LIN {X 0,Y 600.073,Z 913.37,A -85,B 0,C 180,E1 9120.834,E2 9120.834} C_VEL
LIN {X 0,Y 603.97,Z 872.465,A -85,B 0,C 180,E1 9122.572,E2 9122.572} C_VEL
LIN {X 0,Y 605.713,Z 840.651,A -85,B 0,C 180,E1 9123.575,E2 9123.575} C_VEL
LIN {X 0,Y 586.548,Z 799.806,A -85,B 0,C 180,E1 9125.931,E2 9125.931} C_VEL
LIN {X 0,Y 577.288,Z 782.326,A -85,B 0,C 180,E1 9126.944,E2 9126.944} C_VEL
LIN {X 0,Y 577.109,Z 780.81,A -85,B 0,C 180,E1 9127.031,E2 9127.031} C_VEL
LIN {X 0,Y 577.142,Z 780.81,A -85,B 0,C 180,E1 9132.903,E2 9132.903} C_VEL
LIN {X 0,Y 577.108,Z 780.81,A -85,B 0,C 180,E1 9139.116,E2 9139.116} C_VEL
LIN {X 0,Y 577.097,Z 780.81,A -85,B 0,C 180,E1 9144.83,E2 9144.83} C_VEL
LIN {X 0,Y 577.255,Z 780.81,A -85,B 0,C 180,E1 9150.177,E2 9150.177} C_VEL
LIN {X 0,Y 577.406,Z 780.81,A -85,B 0,C 180,E1 9155.248,E2 9155.248} C_VEL
LIN {X 0,Y 577.552,Z 780.81,A -85,B 0,C 180,E1 9160.376,E2 9160.376} C_VEL
LIN {X 0,Y 577.609,Z 780.81,A -85,B 0,C 180,E1 9165.463,E2 9165.463} C_VEL
LIN {X 0,Y 577.862,Z 780.81,A -85,B 0,C 180,E1 9170.972,E2 9170.972} C_VEL
LIN {X 0,Y 578.107,Z 780.81,A -85,B 0,C 180,E1 9177.002,E2 9177.002} C_VEL
LIN {X 0,Y 578.174,Z 780.81,A -85,B 0,C 180,E1 9181.495,E2 9181.495} C_VEL
LIN {X 0,Y 577.898,Z 780.81,A -85,B 0,C 180,E1 9187.509,E2 9187.509} C_VEL
LIN {X 0,Y 577.695,Z 780.81,A -85,B 0,C 180,E1 9193.611,E2 9193.611} C_VEL
LIN {X 0,Y 577.587,Z 780.81,A -85,B 0,C 180,E1 9199.634,E2 9199.634} C_VEL
LIN {X 0,Y 577.399,Z 780.81,A -85,B 0,C 180,E1 9204.748,E2 9204.748} C_VEL
LIN {X 0,Y 577.283,Z 780.81,A -85,B 0,C 180,E1 9210.251,E2 9210.251} C_VEL
LIN {X 0,Y 577.16,Z 780.81,A -85,B 0,C 180,E1 9215.743,E2 9215.743} C_VEL
LIN {X 0,Y 577.065,Z 780.81,A -85,B 0,C 180,E1 9220.882,E2 9220.882} C_VEL
LIN {X 0,Y 577.059,Z 780.81,A -85,B 0,C 180,E1 9227.143,E2 9227.143} C_VEL
LIN {X 0,Y 577.082,Z 780.895,A -85,B 0,C 180,E1 9229.475,E2 9229.475} C_VEL
LIN {X 0,Y 581.683,Z 790.937,A -85,B 0,C 180,E1 9230,E2 9230} C_VEL
LIN {X 0,Y 607.436,Z 841.355,A -85,B 0,C 180,E1 9232.688,E2 9232.688} C_VEL
LIN {X 0,Y 605.125,Z 884.485,A -85,B 0,C 180,E1 9233.623,E2 9233.623} C_VEL
LIN {X 0,Y 604.334,Z 895.912,A -85,B 0,C 180,E1 9233.955,E2 9233.955} C_VEL
LIN {X 0,Y 599.805,Z 912.465,A -85,B 0,C 180,E1 9234.299,E2 9234.299} C_VEL
LIN {X 0,Y 594.958,Z 928.635,A -85,B 0,C 180,E1 9234.736,E2 9234.736} C_VEL
LIN {X 0,Y 590.175,Z 971.895,A -85,B 0,C 180,E1 9236.914,E2 9236.914} C_VEL
LIN {X 0,Y 585.078,Z 1013.237,A -85,B 0,C 180,E1 9239.768,E2 9239.768} C_VEL
LIN {X 0,Y 580.557,Z 1047.846,A -85,B 0,C 180,E1 9242.902,E2 9242.902} C_VEL
LIN {X 0,Y 576.578,Z 1078.993,A -85,B 0,C 180,E1 9246.504,E2 9246.504} C_VEL
LIN {X 0,Y 573.684,Z 1106.248,A -85,B 0,C 180,E1 9250.576,E2 9250.576} C_VEL
LIN {X 0,Y 571.664,Z 1128.837,A -85,B 0,C 180,E1 9255.064,E2 9255.064} C_VEL
LIN {X 0,Y 570.638,Z 1145.24,A -85,B 0,C 180,E1 9259.702,E2 9259.702} C_VEL
LIN {X 0,Y 570.381,Z 1154.482,A -85,B 0,C 180,E1 9263.916,E2 9263.916} C_VEL
LIN {X 0,Y 570.304,Z 1159.165,A -85,B 0,C 180,E1 9268.481,E2 9268.481} C_VEL
LIN {X 0,Y 570.212,Z 1158.218,A -85,B 0,C 180,E1 9273.037,E2 9273.037} C_VEL
LIN {X 0,Y 570.422,Z 1152.885,A -85,B 0,C 180,E1 9277.02,E2 9277.02} C_VEL
LIN {X 0,Y 570.84,Z 1142.468,A -85,B 0,C 180,E1 9281.212,E2 9281.212} C_VEL
LIN {X 0,Y 571.852,Z 1127.098,A -85,B 0,C 180,E1 9285.321,E2 9285.321} C_VEL
LIN {X 0,Y 573.818,Z 1105.125,A -85,B 0,C 180,E1 9289.618,E2 9289.618} C_VEL
LIN {X 0,Y 576.919,Z 1076.481,A -85,B 0,C 180,E1 9293.824,E2 9293.824} C_VEL
LIN {X 0,Y 581.055,Z 1043.921,A -85,B 0,C 180,E1 9297.49,E2 9297.49} C_VEL
LIN {X 0,Y 585.633,Z 1008.232,A -85,B 0,C 180,E1 9300.619,E2 9300.619} C_VEL
LIN {X 0,Y 590.548,Z 969.141,A -85,B 0,C 180,E1 9303.259,E2 9303.259} C_VEL
LIN {X 0,Y 595.375,Z 925.534,A -85,B 0,C 180,E1 9305.435,E2 9305.435} C_VEL
LIN {X 0,Y 599.416,Z 879.277,A -85,B 0,C 180,E1 9307.007,E2 9307.007} C_VEL
LIN {X 0,Y 601.018,Z 843.241,A -85,B 0,C 180,E1 9307.816,E2 9307.816} C_VEL
LIN {X 0,Y 580.212,Z 801.744,A -85,B 0,C 180,E1 9310.177,E2 9310.177} C_VEL
LIN {X 0,Y 569.244,Z 781.517,A -85,B 0,C 180,E1 9311.481,E2 9311.481} C_VEL
LIN {X 0,Y 569.183,Z 780.81,A -85,B 0,C 180,E1 9316.362,E2 9316.362} C_VEL
LIN {X 0,Y 569.222,Z 780.81,A -85,B 0,C 180,E1 9322.379,E2 9322.379} C_VEL
LIN {X 0,Y 569.268,Z 780.81,A -85,B 0,C 180,E1 9328.148,E2 9328.148} C_VEL
LIN {X 0,Y 569.463,Z 780.81,A -85,B 0,C 180,E1 9333.193,E2 9333.193} C_VEL
LIN {X 0,Y 569.555,Z 780.81,A -85,B 0,C 180,E1 9338.215,E2 9338.215} C_VEL
LIN {X 0,Y 569.678,Z 780.81,A -85,B 0,C 180,E1 9343.041,E2 9343.041} C_VEL
LIN {X 0,Y 569.786,Z 780.81,A -85,B 0,C 180,E1 9348.886,E2 9348.886} C_VEL
LIN {X 0,Y 569.989,Z 780.81,A -85,B 0,C 180,E1 9353.916,E2 9353.916} C_VEL
LIN {X 0,Y 570.111,Z 780.81,A -85,B 0,C 180,E1 9358.484,E2 9358.484} C_VEL
LIN {X 0,Y 570.061,Z 780.81,A -85,B 0,C 180,E1 9363.041,E2 9363.041} C_VEL
LIN {X 0,Y 569.988,Z 780.81,A -85,B 0,C 180,E1 9367.618,E2 9367.618} C_VEL
LIN {X 0,Y 569.809,Z 780.81,A -85,B 0,C 180,E1 9372.249,E2 9372.249} C_VEL
LIN {X 0,Y 569.676,Z 780.81,A -85,B 0,C 180,E1 9377.271,E2 9377.271} C_VEL
LIN {X 0,Y 569.524,Z 780.81,A -85,B 0,C 180,E1 9381.804,E2 9381.804} C_VEL
LIN {X 0,Y 569.41,Z 780.81,A -85,B 0,C 180,E1 9386.815,E2 9386.815} C_VEL
LIN {X 0,Y 569.307,Z 780.81,A -85,B 0,C 180,E1 9392.06,E2 9392.06} C_VEL
LIN {X 0,Y 569.177,Z 780.81,A -85,B 0,C 180,E1 9397.63,E2 9397.63} C_VEL
LIN {X 0,Y 569.148,Z 780.81,A -85,B 0,C 180,E1 9403.648,E2 9403.648} C_VEL
LIN {X 0,Y 569.276,Z 780.954,A -85,B 0,C 180,E1 9405.973,E2 9405.973} C_VEL
LIN {X 0,Y 571.747,Z 786.574,A -85,B 0,C 180,E1 9406.291,E2 9406.291} C_VEL
LIN {X 0,Y 592.826,Z 827.014,A -85,B 0,C 180,E1 9408.899,E2 9408.899} C_VEL
LIN {X 0,Y 599.903,Z 845.936,A -85,B 0,C 180,E1 9410.005,E2 9410.005} C_VEL
LIN {X 0,Y 596.272,Z 889.788,A -85,B 0,C 180,E1 9411.521,E2 9411.521} C_VEL
LIN {X 0,Y 591.948,Z 928.384,A -85,B 0,C 180,E1 9413.414,E2 9413.414} C_VEL
LIN {X 0,Y 587.15,Z 967.067,A -85,B 0,C 180,E1 9415.962,E2 9415.962} C_VEL
LIN {X 0,Y 581.942,Z 1004.932,A -85,B 0,C 180,E1 9419.25,E2 9419.25} C_VEL
LIN {X 0,Y 577.433,Z 1037.355,A -85,B 0,C 180,E1 9422.934,E2 9422.934} C_VEL
LIN {X 0,Y 574.125,Z 1065.144,A -85,B 0,C 180,E1 9427.086,E2 9427.086} C_VEL
LIN {X 0,Y 571.998,Z 1085.611,A -85,B 0,C 180,E1 9431.119,E2 9431.119} C_VEL
LIN {X 0,Y 570.903,Z 1101.096,A -85,B 0,C 180,E1 9435.221,E2 9435.221} C_VEL
LIN {X 0,Y 570.424,Z 1111.616,A -85,B 0,C 180,E1 9439.314,E2 9439.314} C_VEL
LIN {X 0,Y 570.232,Z 1116.651,A -85,B 0,C 180,E1 9442.387,E2 9442.387} C_VEL
LIN {X 0,Y 570.235,Z 1119.5,A -85,B 0,C 180,E1 9446.963,E2 9446.963} C_VEL
LIN {X 0,Y 570.363,Z 1116.652,A -85,B 0,C 180,E1 9451.519,E2 9451.519} C_VEL
LIN {X 0,Y 570.477,Z 1110.137,A -85,B 0,C 180,E1 9455.32,E2 9455.32} C_VEL
LIN {X 0,Y 571.138,Z 1096.99,A -85,B 0,C 180,E1 9459.904,E2 9459.904} C_VEL
LIN {X 0,Y 572.65,Z 1079.414,A -85,B 0,C 180,E1 9464.129,E2 9464.129} C_VEL
LIN {X 0,Y 575.037,Z 1056.869,A -85,B 0,C 180,E1 9468.184,E2 9468.184} C_VEL
LIN {X 0,Y 578.775,Z 1027.696,A -85,B 0,C 180,E1 9472.171,E2 9472.171} C_VEL
LIN {X 0,Y 583.598,Z 992.812,A -85,B 0,C 180,E1 9475.807,E2 9475.807} C_VEL
LIN {X 0,Y 588.575,Z 955.332,A -85,B 0,C 180,E1 9478.777,E2 9478.777} C_VEL
LIN {X 0,Y 593.172,Z 916.032,A -85,B 0,C 180,E1 9481.134,E2 9481.134} C_VEL
LIN {X 0,Y 597.321,Z 875.052,A -85,B 0,C 180,E1 9482.926,E2 9482.926} C_VEL
LIN {X 0,Y 599.133,Z 843.251,A -85,B 0,C 180,E1 9483.965,E2 9483.965} C_VEL
LIN {X 0,Y 580.701,Z 803.672,A -85,B 0,C 180,E1 9486.316,E2 9486.316} C_VEL
LIN {X 0,Y 569.37,Z 782.402,A -85,B 0,C 180,E1 9487.595,E2 9487.595} C_VEL
LIN {X 0,Y 569.184,Z 780.81,A -85,B 0,C 180,E1 9487.712,E2 9487.712} C_VEL
LIN {X 0,Y 569.156,Z 780.81,A -85,B 0,C 180,E1 9493.655,E2 9493.655} C_VEL
LIN {X 0,Y 569.128,Z 780.81,A -85,B 0,C 180,E1 9498.417,E2 9498.417} C_VEL
LIN {X 0,Y 569.197,Z 780.81,A -85,B 0,C 180,E1 9504.268,E2 9504.268} C_VEL
LIN {X 0,Y 569.312,Z 780.81,A -85,B 0,C 180,E1 9509.717,E2 9509.717} C_VEL
LIN {X 0,Y 569.463,Z 780.81,A -85,B 0,C 180,E1 9514.879,E2 9514.879} C_VEL
LIN {X 0,Y 569.595,Z 780.81,A -85,B 0,C 180,E1 9519.827,E2 9519.827} C_VEL
LIN {X 0,Y 569.706,Z 780.81,A -85,B 0,C 180,E1 9524.619,E2 9524.619} C_VEL
LIN {X 0,Y 569.835,Z 780.81,A -85,B 0,C 180,E1 9529.302,E2 9529.302} C_VEL
LIN {X 0,Y 570.02,Z 780.81,A -85,B 0,C 180,E1 9533.912,E2 9533.912} C_VEL
LIN {X 0,Y 570.163,Z 780.81,A -85,B 0,C 180,E1 9538.479,E2 9538.479} C_VEL
LIN {X 0,Y 570.058,Z 780.81,A -85,B 0,C 180,E1 9543.036,E2 9543.036} C_VEL
LIN {X 0,Y 569.981,Z 780.81,A -85,B 0,C 180,E1 9547.614,E2 9547.614} C_VEL
LIN {X 0,Y 569.781,Z 780.81,A -85,B 0,C 180,E1 9553.804,E2 9553.804} C_VEL
LIN {X 0,Y 569.669,Z 780.81,A -85,B 0,C 180,E1 9558.555,E2 9558.555} C_VEL
LIN {X 0,Y 569.489,Z 780.81,A -85,B 0,C 180,E1 9563.447,E2 9563.447} C_VEL
LIN {X 0,Y 569.38,Z 780.81,A -85,B 0,C 180,E1 9568.858,E2 9568.858} C_VEL
LIN {X 0,Y 569.276,Z 780.81,A -85,B 0,C 180,E1 9574.625,E2 9574.625} C_VEL
LIN {X 0,Y 569.12,Z 780.81,A -85,B 0,C 180,E1 9579.645,E2 9579.645} C_VEL
LIN {X 0,Y 569.082,Z 780.81,A -85,B 0,C 180,E1 9585.789,E2 9585.789} C_VEL
LIN {X 0,Y 569.135,Z 780.857,A -85,B 0,C 180,E1 9588.819,E2 9588.819} C_VEL
LIN {X 0,Y 573.39,Z 790.326,A -85,B 0,C 180,E1 9589.324,E2 9589.324} C_VEL
LIN {X 0,Y 600.655,Z 843.165,A -85,B 0,C 180,E1 9592.245,E2 9592.245} C_VEL
LIN {X 0,Y 598.252,Z 889.699,A -85,B 0,C 180,E1 9593.337,E2 9593.337} C_VEL
LIN {X 0,Y 594.958,Z 928.635,A -85,B 0,C 180,E1 9594.736,E2 9594.736} C_VEL
LIN {X 0,Y 589.918,Z 944.648,A -85,B 0,C 180,E1 9595.249,E2 9595.249} C_VEL
LIN {X 0,Y 584.727,Z 960.189,A -85,B 0,C 180,E1 9595.838,E2 9595.838} C_VEL
LIN {X 0,Y 579.59,Z 1001.089,A -85,B 0,C 180,E1 9598.448,E2 9598.448} C_VEL
LIN {X 0,Y 574.319,Z 1039.727,A -85,B 0,C 180,E1 9601.731,E2 9601.731} C_VEL
LIN {X 0,Y 569.837,Z 1073.683,A -85,B 0,C 180,E1 9605.521,E2 9605.521} C_VEL
LIN {X 0,Y 566.452,Z 1101.165,A -85,B 0,C 180,E1 9609.497,E2 9609.497} C_VEL
LIN {X 0,Y 564.329,Z 1123.284,A -85,B 0,C 180,E1 9613.67,E2 9613.67} C_VEL
LIN {X 0,Y 562.989,Z 1140.694,A -85,B 0,C 180,E1 9618.131,E2 9618.131} C_VEL
LIN {X 0,Y 562.565,Z 1151.534,A -85,B 0,C 180,E1 9622.281,E2 9622.281} C_VEL
LIN {X 0,Y 562.366,Z 1156.624,A -85,B 0,C 180,E1 9625.375,E2 9625.375} C_VEL
LIN {X 0,Y 562.351,Z 1159.5,A -85,B 0,C 180,E1 9629.999,E2 9629.999} C_VEL
LIN {X 0,Y 562.352,Z 1156.627,A -85,B 0,C 180,E1 9634.623,E2 9634.623} C_VEL
LIN {X 0,Y 562.612,Z 1149.938,A -85,B 0,C 180,E1 9638.494,E2 9638.494} C_VEL
LIN {X 0,Y 563.221,Z 1137.519,A -85,B 0,C 180,E1 9642.787,E2 9642.787} C_VEL
LIN {X 0,Y 564.536,Z 1119.557,A -85,B 0,C 180,E1 9647.123,E2 9647.123} C_VEL
LIN {X 0,Y 567.089,Z 1095.365,A -85,B 0,C 180,E1 9651.441,E2 9651.441} C_VEL
LIN {X 0,Y 571.046,Z 1063.857,A -85,B 0,C 180,E1 9655.681,E2 9655.681} C_VEL
LIN {X 0,Y 576.012,Z 1028.064,A -85,B 0,C 180,E1 9659.356,E2 9659.356} C_VEL
LIN {X 0,Y 581.404,Z 988.132,A -85,B 0,C 180,E1 9662.483,E2 9662.483} C_VEL
LIN {X 0,Y 586.519,Z 947.561,A -85,B 0,C 180,E1 9664.855,E2 9664.855} C_VEL
LIN {X 0,Y 590.785,Z 906.842,A -85,B 0,C 180,E1 9666.603,E2 9666.603} C_VEL
LIN {X 0,Y 594.315,Z 862.108,A -85,B 0,C 180,E1 9667.891,E2 9667.891} C_VEL
LIN {X 0,Y 594.726,Z 845.916,A -85,B 0,C 180,E1 9668.246,E2 9668.246} C_VEL
LIN {X 0,Y 574.568,Z 805.711,A -85,B 0,C 180,E1 9670.603,E2 9670.603} C_VEL
LIN {X 0,Y 561.378,Z 781.906,A -85,B 0,C 180,E1 9672.211,E2 9672.211} C_VEL
LIN {X 0,Y 561.272,Z 780.81,A -85,B 0,C 180,E1 9672.303,E2 9672.303} C_VEL
LIN {X 0,Y 561.238,Z 780.81,A -85,B 0,C 180,E1 9677.704,E2 9677.704} C_VEL
LIN {X 0,Y 561.303,Z 780.81,A -85,B 0,C 180,E1 9683.865,E2 9683.865} C_VEL
LIN {X 0,Y 561.396,Z 780.81,A -85,B 0,C 180,E1 9689.466,E2 9689.466} C_VEL
LIN {X 0,Y 561.567,Z 780.81,A -85,B 0,C 180,E1 9694.505,E2 9694.505} C_VEL
LIN {X 0,Y 561.662,Z 780.81,A -85,B 0,C 180,E1 9700.327,E2 9700.327} C_VEL
LIN {X 0,Y 561.785,Z 780.81,A -85,B 0,C 180,E1 9705.995,E2 9705.995} C_VEL
LIN {X 0,Y 561.988,Z 780.81,A -85,B 0,C 180,E1 9710.72,E2 9710.72} C_VEL
LIN {X 0,Y 562.269,Z 780.81,A -85,B 0,C 180,E1 9716.922,E2 9716.922} C_VEL
LIN {X 0,Y 562.343,Z 780.81,A -85,B 0,C 180,E1 9721.542,E2 9721.542} C_VEL
LIN {X 0,Y 562.078,Z 780.81,A -85,B 0,C 180,E1 9727.726,E2 9727.726} C_VEL
LIN {X 0,Y 561.886,Z 780.81,A -85,B 0,C 180,E1 9732.424,E2 9732.424} C_VEL
LIN {X 0,Y 561.778,Z 780.81,A -85,B 0,C 180,E1 9737.21,E2 9737.21} C_VEL
LIN {X 0,Y 561.573,Z 780.81,A -85,B 0,C 180,E1 9742.129,E2 9742.129} C_VEL
LIN {X 0,Y 561.46,Z 780.81,A -85,B 0,C 180,E1 9747.36,E2 9747.36} C_VEL
LIN {X 0,Y 561.329,Z 780.81,A -85,B 0,C 180,E1 9752.571,E2 9752.571} C_VEL
LIN {X 0,Y 561.195,Z 780.81,A -85,B 0,C 180,E1 9758.261,E2 9758.261} C_VEL
LIN {X 0,Y 561.275,Z 780.81,A -85,B 0,C 180,E1 9764.42,E2 9764.42} C_VEL
LIN {X 0,Y 561.322,Z 780.982,A -85,B 0,C 180,E1 9765.228,E2 9765.228} C_VEL
LIN {X 0,Y 563.735,Z 786.436,A -85,B 0,C 180,E1 9765.55,E2 9765.55} C_VEL
LIN {X 0,Y 585.464,Z 827.456,A -85,B 0,C 180,E1 9768.315,E2 9768.315} C_VEL
LIN {X 0,Y 593.533,Z 847.958,A -85,B 0,C 180,E1 9769.588,E2 9769.588} C_VEL
LIN {X 0,Y 589.521,Z 893.333,A -85,B 0,C 180,E1 9771.197,E2 9771.197} C_VEL
LIN {X 0,Y 584.562,Z 936.072,A -85,B 0,C 180,E1 9773.413,E2 9773.413} C_VEL
LIN {X 0,Y 579.253,Z 974.509,A -85,B 0,C 180,E1 9776.11,E2 9776.11} C_VEL
LIN {X 0,Y 574.2,Z 1009.101,A -85,B 0,C 180,E1 9779.279,E2 9779.279} C_VEL
LIN {X 0,Y 569.854,Z 1039.146,A -85,B 0,C 180,E1 9782.804,E2 9782.804} C_VEL
LIN {X 0,Y 566.476,Z 1065.895,A -85,B 0,C 180,E1 9786.885,E2 9786.885} C_VEL
LIN {X 0,Y 564.137,Z 1087.43,A -85,B 0,C 180,E1 9791.251,E2 9791.251} C_VEL
LIN {X 0,Y 562.983,Z 1102.705,A -85,B 0,C 180,E1 9795.515,E2 9795.515} C_VEL
LIN {X 0,Y 562.49,Z 1113.256,A -85,B 0,C 180,E1 9799.944,E2 9799.944} C_VEL
LIN {X 0,Y 562.254,Z 1118.267,A -85,B 0,C 180,E1 9803.867,E2 9803.867} C_VEL
LIN {X 0,Y 562.251,Z 1119.209,A -85,B 0,C 180,E1 9808.461,E2 9808.461} C_VEL
LIN {X 0,Y 562.475,Z 1114.665,A -85,B 0,C 180,E1 9813.081,E2 9813.081} C_VEL
LIN {X 0,Y 562.856,Z 1106.581,A -85,B 0,C 180,E1 9817.009,E2 9817.009} C_VEL
LIN {X 0,Y 563.809,Z 1092.172,A -85,B 0,C 180,E1 9821.475,E2 9821.475} C_VEL
LIN {X 0,Y 565.609,Z 1072.68,A -85,B 0,C 180,E1 9825.776,E2 9825.776} C_VEL
LIN {X 0,Y 568.828,Z 1047.041,A -85,B 0,C 180,E1 9830.002,E2 9830.002} C_VEL
LIN {X 0,Y 573.203,Z 1016.141,A -85,B 0,C 180,E1 9833.881,E2 9833.881} C_VEL
LIN {X 0,Y 578.477,Z 979.558,A -85,B 0,C 180,E1 9837.372,E2 9837.372} C_VEL
LIN {X 0,Y 583.722,Z 940.551,A -85,B 0,C 180,E1 9840.179,E2 9840.179} C_VEL
LIN {X 0,Y 588.242,Z 901.026,A -85,B 0,C 180,E1 9842.308,E2 9842.308} C_VEL
LIN {X 0,Y 592.238,Z 857.862,A -85,B 0,C 180,E1 9843.962,E2 9843.962} C_VEL
LIN {X 0,Y 592.521,Z 845.7,A -85,B 0,C 180,E1 9844.366,E2 9844.366} C_VEL
LIN {X 0,Y 574.238,Z 806.125,A -85,B 0,C 180,E1 9846.787,E2 9846.787} C_VEL
LIN {X 0,Y 561.498,Z 782.258,A -85,B 0,C 180,E1 9848.269,E2 9848.269} C_VEL
LIN {X 0,Y 561.339,Z 780.81,A -85,B 0,C 180,E1 9848.378,E2 9848.378} C_VEL
LIN {X 0,Y 561.265,Z 780.81,A -85,B 0,C 180,E1 9854.428,E2 9854.428} C_VEL
LIN {X 0,Y 561.187,Z 780.81,A -85,B 0,C 180,E1 9859.746,E2 9859.746} C_VEL
LIN {X 0,Y 561.286,Z 780.81,A -85,B 0,C 180,E1 9865.576,E2 9865.576} C_VEL
LIN {X 0,Y 561.458,Z 780.81,A -85,B 0,C 180,E1 9871.026,E2 9871.026} C_VEL
LIN {X 0,Y 561.555,Z 780.81,A -85,B 0,C 180,E1 9876.196,E2 9876.196} C_VEL
LIN {X 0,Y 561.71,Z 780.81,A -85,B 0,C 180,E1 9881.167,E2 9881.167} C_VEL
LIN {X 0,Y 561.788,Z 780.81,A -85,B 0,C 180,E1 9885.991,E2 9885.991} C_VEL
LIN {X 0,Y 562.022,Z 780.81,A -85,B 0,C 180,E1 9890.716,E2 9890.716} C_VEL
LIN {X 0,Y 562.29,Z 780.81,A -85,B 0,C 180,E1 9896.917,E2 9896.917} C_VEL
LIN {X 0,Y 562.359,Z 780.81,A -85,B 0,C 180,E1 9901.537,E2 9901.537} C_VEL
LIN {X 0,Y 562.072,Z 780.81,A -85,B 0,C 180,E1 9907.722,E2 9907.722} C_VEL
LIN {X 0,Y 561.879,Z 780.81,A -85,B 0,C 180,E1 9912.42,E2 9912.42} C_VEL
LIN {X 0,Y 561.801,Z 780.81,A -85,B 0,C 180,E1 9917.204,E2 9917.204} C_VEL
LIN {X 0,Y 561.62,Z 780.81,A -85,B 0,C 180,E1 9922.122,E2 9922.122} C_VEL
LIN {X 0,Y 561.511,Z 780.81,A -85,B 0,C 180,E1 9927.366,E2 9927.366} C_VEL
LIN {X 0,Y 561.392,Z 780.81,A -85,B 0,C 180,E1 9932.562,E2 9932.562} C_VEL
LIN {X 0,Y 561.218,Z 780.81,A -85,B 0,C 180,E1 9938.253,E2 9938.253} C_VEL
LIN {X 0,Y 561.157,Z 780.81,A -85,B 0,C 180,E1 9944.425,E2 9944.425} C_VEL
LIN {X 0,Y 561.21,Z 781.002,A -85,B 0,C 180,E1 9948.144,E2 9948.144} C_VEL
LIN {X 0,Y 565.518,Z 790.341,A -85,B 0,C 180,E1 9948.667,E2 9948.667} C_VEL
LIN {X 0,Y 593.173,Z 843.528,A -85,B 0,C 180,E1 9951.713,E2 9951.713} C_VEL
LIN {X 0,Y 594.62,Z 848.331,A -85,B 0,C 180,E1 9951.919,E2 9951.919} C_VEL
LIN {X 0,Y 591.458,Z 893.931,A -85,B 0,C 180,E1 9953.016,E2 9953.016} C_VEL
LIN {X 0,Y 587.442,Z 937.061,A -85,B 0,C 180,E1 9954.685,E2 9954.685} C_VEL
LIN {X 0,Y 584.727,Z 960.189,A -85,B 0,C 180,E1 9955.838,E2 9955.838} C_VEL
LIN {X 0,Y 579.417,Z 975.478,A -85,B 0,C 180,E1 9956.52,E2 9956.52} C_VEL
LIN {X 0,Y 574.12,Z 990.222,A -85,B 0,C 180,E1 9957.283,E2 9957.283} C_VEL
LIN {X 0,Y 568.731,Z 1028.734,A -85,B 0,C 180,E1 9960.338,E2 9960.338} C_VEL
LIN {X 0,Y 563.617,Z 1063.889,A -85,B 0,C 180,E1 9963.988,E2 9963.988} C_VEL
LIN {X 0,Y 559.514,Z 1094.68,A -85,B 0,C 180,E1 9968.186,E2 9968.186} C_VEL
LIN {X 0,Y 556.807,Z 1119.288,A -85,B 0,C 180,E1 9972.63,E2 9972.63} C_VEL
LIN {X 0,Y 555.36,Z 1137.235,A -85,B 0,C 180,E1 9977.027,E2 9977.027} C_VEL
LIN {X 0,Y 554.735,Z 1149.655,A -85,B 0,C 180,E1 9981.383,E2 9981.383} C_VEL
LIN {X 0,Y 554.492,Z 1156.344,A -85,B 0,C 180,E1 9985.31,E2 9985.31} C_VEL
LIN {X 0,Y 554.469,Z 1159.251,A -85,B 0,C 180,E1 9989.999,E2 9989.999} C_VEL
LIN {X 0,Y 554.479,Z 1156.345,A -85,B 0,C 180,E1 9994.689,E2 9994.689} C_VEL
LIN {X 0,Y 554.725,Z 1149.652,A -85,B 0,C 180,E1 9998.616,E2 9998.616} C_VEL
LIN {X 0,Y 555.354,Z 1137.229,A -85,B 0,C 180,E1 10002.971,E2 10002.971} C_VEL
LIN {X 0,Y 556.621,Z 1121.205,A -85,B 0,C 180,E1 10006.967,E2 10006.967} C_VEL
LIN {X 0,Y 559.203,Z 1097.141,A -85,B 0,C 180,E1 10011.408,E2 10011.408} C_VEL
LIN {X 0,Y 562.974,Z 1068.487,A -85,B 0,C 180,E1 10015.432,E2 10015.432} C_VEL
LIN {X 0,Y 567.604,Z 1036.311,A -85,B 0,C 180,E1 10018.959,E2 10018.959} C_VEL
LIN {X 0,Y 573.103,Z 998.779,A -85,B 0,C 180,E1 10022.146,E2 10022.146} C_VEL
LIN {X 0,Y 578.792,Z 957.096,A -85,B 0,C 180,E1 10024.812,E2 10024.812} C_VEL
LIN {X 0,Y 583.798,Z 912.757,A -85,B 0,C 180,E1 10026.857,E2 10026.857} C_VEL
LIN {X 0,Y 587.711,Z 867.328,A -85,B 0,C 180,E1 10028.246,E2 10028.246} C_VEL
LIN {X 0,Y 588.397,Z 848.496,A -85,B 0,C 180,E1 10028.681,E2 10028.681} C_VEL
LIN {X 0,Y 568.062,Z 807.724,A -85,B 0,C 180,E1 10031.152,E2 10031.152} C_VEL
LIN {X 0,Y 553.51,Z 782.184,A -85,B 0,C 180,E1 10032.974,E2 10032.974} C_VEL
LIN {X 0,Y 553.388,Z 780.81,A -85,B 0,C 180,E1 10033.051,E2 10033.051} C_VEL
LIN {X 0,Y 553.313,Z 780.81,A -85,B 0,C 180,E1 10039.058,E2 10039.058} C_VEL
LIN {X 0,Y 553.36,Z 780.81,A -85,B 0,C 180,E1 10045.018,E2 10045.018} C_VEL
LIN {X 0,Y 553.555,Z 780.81,A -85,B 0,C 180,E1 10050.871,E2 10050.871} C_VEL
LIN {X 0,Y 553.646,Z 780.81,A -85,B 0,C 180,E1 10055.84,E2 10055.84} C_VEL
LIN {X 0,Y 553.797,Z 780.81,A -85,B 0,C 180,E1 10060.893,E2 10060.893} C_VEL
LIN {X 0,Y 553.883,Z 780.81,A -85,B 0,C 180,E1 10065.791,E2 10065.791} C_VEL
LIN {X 0,Y 554.064,Z 780.81,A -85,B 0,C 180,E1 10070.586,E2 10070.586} C_VEL
LIN {X 0,Y 554.238,Z 780.81,A -85,B 0,C 180,E1 10075.312,E2 10075.312} C_VEL
LIN {X 0,Y 554.473,Z 780.81,A -85,B 0,C 180,E1 10080.002,E2 10080.002} C_VEL
LIN {X 0,Y 554.234,Z 780.81,A -85,B 0,C 180,E1 10086.262,E2 10086.262} C_VEL
LIN {X 0,Y 554.028,Z 780.81,A -85,B 0,C 180,E1 10091.007,E2 10091.007} C_VEL
LIN {X 0,Y 553.886,Z 780.81,A -85,B 0,C 180,E1 10095.832,E2 10095.832} C_VEL
LIN {X 0,Y 553.704,Z 780.81,A -85,B 0,C 180,E1 10100.779,E2 10100.779} C_VEL
LIN {X 0,Y 553.565,Z 780.81,A -85,B 0,C 180,E1 10105.895,E2 10105.895} C_VEL
LIN {X 0,Y 553.427,Z 780.81,A -85,B 0,C 180,E1 10111.248,E2 10111.248} C_VEL
LIN {X 0,Y 553.295,Z 780.81,A -85,B 0,C 180,E1 10116.926,E2 10116.926} C_VEL
LIN {X 0,Y 553.319,Z 780.81,A -85,B 0,C 180,E1 10123.053,E2 10123.053} C_VEL
LIN {X 0,Y 553.399,Z 781.312,A -85,B 0,C 180,E1 10124.461,E2 10124.461} C_VEL
LIN {X 0,Y 558.698,Z 791.551,A -85,B 0,C 180,E1 10125.159,E2 10125.159} C_VEL
LIN {X 0,Y 578.749,Z 829.202,A -85,B 0,C 180,E1 10127.798,E2 10127.798} C_VEL
LIN {X 0,Y 587.053,Z 850.937,A -85,B 0,C 180,E1 10129.184,E2 10129.184} C_VEL
LIN {X 0,Y 583.038,Z 894.618,A -85,B 0,C 180,E1 10130.776,E2 10130.776} C_VEL
LIN {X 0,Y 577.853,Z 937.393,A -85,B 0,C 180,E1 10133.027,E2 10133.027} C_VEL
LIN {X 0,Y 572.095,Z 976.893,A -85,B 0,C 180,E1 10135.856,E2 10135.856} C_VEL
LIN {X 0,Y 566.781,Z 1011.24,A -85,B 0,C 180,E1 10139.09,E2 10139.09} C_VEL
LIN {X 0,Y 562.37,Z 1040.071,A -85,B 0,C 180,E1 10142.554,E2 10142.554} C_VEL
LIN {X 0,Y 558.73,Z 1067.555,A -85,B 0,C 180,E1 10146.842,E2 10146.842} C_VEL
LIN {X 0,Y 556.234,Z 1089.902,A -85,B 0,C 180,E1 10151.544,E2 10151.544} C_VEL
LIN {X 0,Y 555.047,Z 1105.446,A -85,B 0,C 180,E1 10156.22,E2 10156.22} C_VEL
LIN {X 0,Y 554.545,Z 1114.728,A -85,B 0,C 180,E1 10160.591,E2 10160.591} C_VEL
LIN {X 0,Y 554.342,Z 1119.448,A -85,B 0,C 180,E1 10165.31,E2 10165.31} C_VEL
LIN {X 0,Y 554.512,Z 1118.579,A -85,B 0,C 180,E1 10170.001,E2 10170.001} C_VEL
LIN {X 0,Y 554.716,Z 1113.829,A -85,B 0,C 180,E1 10173.906,E2 10173.906} C_VEL
LIN {X 0,Y 555.148,Z 1102.828,A -85,B 0,C 180,E1 10178.611,E2 10178.611} C_VEL
LIN {X 0,Y 556.478,Z 1087.415,A -85,B 0,C 180,E1 10182.947,E2 10182.947} C_VEL
LIN {X 0,Y 558.854,Z 1066.18,A -85,B 0,C 180,E1 10187.304,E2 10187.304} C_VEL
LIN {X 0,Y 562.56,Z 1039.173,A -85,B 0,C 180,E1 10191.469,E2 10191.469} C_VEL
LIN {X 0,Y 567.374,Z 1007.213,A -85,B 0,C 180,E1 10195.223,E2 10195.223} C_VEL
LIN {X 0,Y 572.54,Z 972.464,A -85,B 0,C 180,E1 10198.365,E2 10198.365} C_VEL
LIN {X 0,Y 577.825,Z 934.567,A -85,B 0,C 180,E1 10200.989,E2 10200.989} C_VEL
LIN {X 0,Y 582.618,Z 893.616,A -85,B 0,C 180,E1 10203.1,E2 10203.1} C_VEL
LIN {X 0,Y 586.033,Z 848.57,A -85,B 0,C 180,E1 10204.744,E2 10204.744} C_VEL
LIN {X 0,Y 568.415,Z 809.937,A -85,B 0,C 180,E1 10207.193,E2 10207.193} C_VEL
LIN {X 0,Y 553.505,Z 782.173,A -85,B 0,C 180,E1 10208.979,E2 10208.979} C_VEL
LIN {X 0,Y 553.345,Z 780.81,A -85,B 0,C 180,E1 10209.162,E2 10209.162} C_VEL
LIN {X 0,Y 553.359,Z 780.81,A -85,B 0,C 180,E1 10215.237,E2 10215.237} C_VEL
LIN {X 0,Y 553.264,Z 780.81,A -85,B 0,C 180,E1 10221.088,E2 10221.088} C_VEL
LIN {X 0,Y 553.353,Z 780.81,A -85,B 0,C 180,E1 10226.899,E2 10226.899} C_VEL
LIN {X 0,Y 553.578,Z 780.81,A -85,B 0,C 180,E1 10232.354,E2 10232.354} C_VEL
LIN {X 0,Y 553.691,Z 780.81,A -85,B 0,C 180,E1 10238.114,E2 10238.114} C_VEL
LIN {X 0,Y 553.874,Z 780.81,A -85,B 0,C 180,E1 10242.727,E2 10242.727} C_VEL
LIN {X 0,Y 554.03,Z 780.81,A -85,B 0,C 180,E1 10249.084,E2 10249.084} C_VEL
LIN {X 0,Y 554.205,Z 780.81,A -85,B 0,C 180,E1 10253.737,E2 10253.737} C_VEL
LIN {X 0,Y 554.367,Z 780.81,A -85,B 0,C 180,E1 10258.436,E2 10258.436} C_VEL
LIN {X 0,Y 554.25,Z 780.81,A -85,B 0,C 180,E1 10263.123,E2 10263.123} C_VEL
LIN {X 0,Y 554.154,Z 780.81,A -85,B 0,C 180,E1 10267.833,E2 10267.833} C_VEL
LIN {X 0,Y 553.969,Z 780.81,A -85,B 0,C 180,E1 10272.6,E2 10272.6} C_VEL
LIN {X 0,Y 553.877,Z 780.81,A -85,B 0,C 180,E1 10277.458,E2 10277.458} C_VEL
LIN {X 0,Y 553.691,Z 780.81,A -85,B 0,C 180,E1 10282.456,E2 10282.456} C_VEL
LIN {X 0,Y 553.585,Z 780.81,A -85,B 0,C 180,E1 10287.641,E2 10287.641} C_VEL
LIN {X 0,Y 553.463,Z 780.81,A -85,B 0,C 180,E1 10293.088,E2 10293.088} C_VEL
LIN {X 0,Y 553.269,Z 780.81,A -85,B 0,C 180,E1 10298.905,E2 10298.905} C_VEL
LIN {X 0,Y 553.275,Z 780.81,A -85,B 0,C 180,E1 10305.231,E2 10305.231} C_VEL
LIN {X 0,Y 553.231,Z 780.81,A -85,B 0,C 180,E1 10307.425,E2 10307.425} C_VEL
LIN {X 0,Y 557.458,Z 790.088,A -85,B 0,C 180,E1 10307.965,E2 10307.965} C_VEL
LIN {X 0,Y 584.395,Z 841.117,A -85,B 0,C 180,E1 10311.017,E2 10311.017} C_VEL
LIN {X 0,Y 588.113,Z 850.932,A -85,B 0,C 180,E1 10311.505,E2 10311.505} C_VEL
LIN {X 0,Y 584.853,Z 895.964,A -85,B 0,C 180,E1 10312.632,E2 10312.632} C_VEL
LIN {X 0,Y 580.623,Z 938.923,A -85,B 0,C 180,E1 10314.335,E2 10314.335} C_VEL
LIN {X 0,Y 575.55,Z 979.018,A -85,B 0,C 180,E1 10316.539,E2 10316.539} C_VEL
LIN {X 0,Y 574.12,Z 990.222,A -85,B 0,C 180,E1 10317.283,E2 10317.283} C_VEL
LIN {X 0,Y 568.609,Z 1004.63,A -85,B 0,C 180,E1 10318.131,E2 10318.131} C_VEL
LIN {X 0,Y 563.059,Z 1018.466,A -85,B 0,C 180,E1 10319.056,E2 10319.056} C_VEL
LIN {X 0,Y 557.878,Z 1053.087,A -85,B 0,C 180,E1 10322.418,E2 10322.418} C_VEL
LIN {X 0,Y 553.212,Z 1084.677,A -85,B 0,C 180,E1 10326.399,E2 10326.399} C_VEL
LIN {X 0,Y 549.979,Z 1110.894,A -85,B 0,C 180,E1 10330.748,E2 10330.748} C_VEL
LIN {X 0,Y 548.01,Z 1130.906,A -85,B 0,C 180,E1 10335.17,E2 10335.17} C_VEL
LIN {X 0,Y 547.003,Z 1145.474,A -85,B 0,C 180,E1 10339.655,E2 10339.655} C_VEL
LIN {X 0,Y 546.697,Z 1154.662,A -85,B 0,C 180,E1 10344.182,E2 10344.182} C_VEL
LIN {X 0,Y 546.626,Z 1158.63,A -85,B 0,C 180,E1 10348.415,E2 10348.415} C_VEL
LIN {X 0,Y 546.534,Z 1157.655,A -85,B 0,C 180,E1 10353.169,E2 10353.169} C_VEL
LIN {X 0,Y 546.732,Z 1152.56,A -85,B 0,C 180,E1 10357.144,E2 10357.144} C_VEL
LIN {X 0,Y 547.258,Z 1141.531,A -85,B 0,C 180,E1 10361.726,E2 10361.726} C_VEL
LIN {X 0,Y 548.45,Z 1126.22,A -85,B 0,C 180,E1 10365.992,E2 10365.992} C_VEL
LIN {X 0,Y 550.714,Z 1104.231,A -85,B 0,C 180,E1 10370.477,E2 10370.477} C_VEL
LIN {X 0,Y 554.687,Z 1074.687,A -85,B 0,C 180,E1 10374.976,E2 10374.976} C_VEL
LIN {X 0,Y 560.073,Z 1039.291,A -85,B 0,C 180,E1 10379.054,E2 10379.054} C_VEL
LIN {X 0,Y 565.975,Z 1000.59,A -85,B 0,C 180,E1 10382.44,E2 10382.44} C_VEL
LIN {X 0,Y 571.977,Z 958.626,A -85,B 0,C 180,E1 10385.181,E2 10385.181} C_VEL
LIN {X 0,Y 577.106,Z 915.926,A -85,B 0,C 180,E1 10387.206,E2 10387.206} C_VEL
LIN {X 0,Y 581.188,Z 872.434,A -85,B 0,C 180,E1 10388.608,E2 10388.608} C_VEL
LIN {X 0,Y 582.147,Z 851.273,A -85,B 0,C 180,E1 10389.117,E2 10389.117} C_VEL
LIN {X 0,Y 562.499,Z 811.672,A -85,B 0,C 180,E1 10391.597,E2 10391.597} C_VEL
LIN {X 0,Y 545.528,Z 781.841,A -85,B 0,C 180,E1 10393.793,E2 10393.793} C_VEL
LIN {X 0,Y 545.433,Z 780.81,A -85,B 0,C 180,E1 10393.933,E2 10393.933} C_VEL
LIN {X 0,Y 545.389,Z 780.81,A -85,B 0,C 180,E1 10400.424,E2 10400.424} C_VEL
LIN {X 0,Y 545.396,Z 780.81,A -85,B 0,C 180,E1 10406.359,E2 10406.359} C_VEL
LIN {X 0,Y 545.673,Z 780.81,A -85,B 0,C 180,E1 10412.393,E2 10412.393} C_VEL
LIN {X 0,Y 545.726,Z 780.81,A -85,B 0,C 180,E1 10417.198,E2 10417.198} C_VEL
LIN {X 0,Y 545.881,Z 780.81,A -85,B 0,C 180,E1 10422.278,E2 10422.278} C_VEL
LIN {X 0,Y 545.996,Z 780.81,A -85,B 0,C 180,E1 10427.213,E2 10427.213} C_VEL
LIN {X 0,Y 546.243,Z 780.81,A -85,B 0,C 180,E1 10432.053,E2 10432.053} C_VEL
LIN {X 0,Y 546.449,Z 780.81,A -85,B 0,C 180,E1 10436.833,E2 10436.833} C_VEL
LIN {X 0,Y 546.533,Z 780.81,A -85,B 0,C 180,E1 10441.587,E2 10441.587} C_VEL
LIN {X 0,Y 546.348,Z 780.81,A -85,B 0,C 180,E1 10446.353,E2 10446.353} C_VEL
LIN {X 0,Y 546.103,Z 780.81,A -85,B 0,C 180,E1 10451.169,E2 10451.169} C_VEL
LIN {X 0,Y 545.96,Z 780.81,A -85,B 0,C 180,E1 10456.068,E2 10456.068} C_VEL
LIN {X 0,Y 545.776,Z 780.81,A -85,B 0,C 180,E1 10461.095,E2 10461.095} C_VEL
LIN {X 0,Y 545.613,Z 780.81,A -85,B 0,C 180,E1 10466.302,E2 10466.302} C_VEL
LIN {X 0,Y 545.494,Z 780.81,A -85,B 0,C 180,E1 10471.755,E2 10471.755} C_VEL
LIN {X 0,Y 545.385,Z 780.81,A -85,B 0,C 180,E1 10477.553,E2 10477.553} C_VEL
LIN {X 0,Y 545.415,Z 780.81,A -85,B 0,C 180,E1 10483.635,E2 10483.635} C_VEL
LIN {X 0,Y 547.646,Z 786.298,A -85,B 0,C 180,E1 10483.968,E2 10483.968} C_VEL
LIN {X 0,Y 569.01,Z 824.763,A -85,B 0,C 180,E1 10486.836,E2 10486.836} C_VEL
LIN {X 0,Y 580.741,Z 853.326,A -85,B 0,C 180,E1 10488.76,E2 10488.76} C_VEL
LIN {X 0,Y 576.508,Z 896.529,A -85,B 0,C 180,E1 10490.374,E2 10490.374} C_VEL
LIN {X 0,Y 571.164,Z 938.52,A -85,B 0,C 180,E1 10492.619,E2 10492.619} C_VEL
LIN {X 0,Y 565.074,Z 978.442,A -85,B 0,C 180,E1 10495.527,E2 10495.527} C_VEL
LIN {X 0,Y 559.276,Z 1014.12,A -85,B 0,C 180,E1 10498.975,E2 10498.975} C_VEL
LIN {X 0,Y 554.573,Z 1043.311,A -85,B 0,C 180,E1 10502.626,E2 10502.626} C_VEL
LIN {X 0,Y 551.004,Z 1068.771,A -85,B 0,C 180,E1 10506.73,E2 10506.73} C_VEL
LIN {X 0,Y 548.505,Z 1089.734,A -85,B 0,C 180,E1 10511.209,E2 10511.209} C_VEL
LIN {X 0,Y 547.269,Z 1104.472,A -85,B 0,C 180,E1 10515.612,E2 10515.612} C_VEL
LIN {X 0,Y 546.748,Z 1113.652,A -85,B 0,C 180,E1 10519.652,E2 10519.652} C_VEL
LIN {X 0,Y 546.467,Z 1118.737,A -85,B 0,C 180,E1 10523.65,E2 10523.65} C_VEL
LIN {X 0,Y 546.544,Z 1120.05,A -85,B 0,C 180,E1 10526.831,E2 10526.831} C_VEL
LIN {X 0,Y 546.699,Z 1117.418,A -85,B 0,C 180,E1 10531.585,E2 10531.585} C_VEL
LIN {X 0,Y 546.931,Z 1110.188,A -85,B 0,C 180,E1 10536.008,E2 10536.008} C_VEL
LIN {X 0,Y 547.89,Z 1096.974,A -85,B 0,C 180,E1 10540.73,E2 10540.73} C_VEL
LIN {X 0,Y 549.708,Z 1079.018,A -85,B 0,C 180,E1 10545.139,E2 10545.139} C_VEL
LIN {X 0,Y 552.712,Z 1055.865,A -85,B 0,C 180,E1 10549.385,E2 10549.385} C_VEL
LIN {X 0,Y 557.084,Z 1027.357,A -85,B 0,C 180,E1 10553.373,E2 10553.373} C_VEL
LIN {X 0,Y 562.61,Z 992.773,A -85,B 0,C 180,E1 10557.061,E2 10557.061} C_VEL
LIN {X 0,Y 568.61,Z 953.202,A -85,B 0,C 180,E1 10560.243,E2 10560.243} C_VEL
LIN {X 0,Y 574.016,Z 911.262,A -85,B 0,C 180,E1 10562.744,E2 10562.744} C_VEL
LIN {X 0,Y 578.662,Z 867.789,A -85,B 0,C 180,E1 10564.573,E2 10564.573} C_VEL
LIN {X 0,Y 579.477,Z 851.147,A -85,B 0,C 180,E1 10565.149,E2 10565.149} C_VEL
LIN {X 0,Y 561.702,Z 811.844,A -85,B 0,C 180,E1 10567.721,E2 10567.721} C_VEL
LIN {X 0,Y 545.432,Z 781.534,A -85,B 0,C 180,E1 10569.735,E2 10569.735} C_VEL
LIN {X 0,Y 545.384,Z 780.81,A -85,B 0,C 180,E1 10573.92,E2 10573.92} C_VEL
LIN {X 0,Y 545.355,Z 780.81,A -85,B 0,C 180,E1 10580.414,E2 10580.414} C_VEL
LIN {X 0,Y 545.391,Z 780.81,A -85,B 0,C 180,E1 10586.352,E2 10586.352} C_VEL
LIN {X 0,Y 545.679,Z 780.81,A -85,B 0,C 180,E1 10592.395,E2 10592.395} C_VEL
LIN {X 0,Y 545.722,Z 780.81,A -85,B 0,C 180,E1 10597.193,E2 10597.193} C_VEL
LIN {X 0,Y 545.903,Z 780.81,A -85,B 0,C 180,E1 10602.273,E2 10602.273} C_VEL
LIN {X 0,Y 546.014,Z 780.81,A -85,B 0,C 180,E1 10607.208,E2 10607.208} C_VEL
LIN {X 0,Y 546.239,Z 780.81,A -85,B 0,C 180,E1 10613.105,E2 10613.105} C_VEL
LIN {X 0,Y 546.465,Z 780.81,A -85,B 0,C 180,E1 10618.413,E2 10618.413} C_VEL
LIN {X 0,Y 546.346,Z 780.81,A -85,B 0,C 180,E1 10623.168,E2 10623.168} C_VEL
LIN {X 0,Y 546.247,Z 780.81,A -85,B 0,C 180,E1 10627.947,E2 10627.947} C_VEL
LIN {X 0,Y 546.044,Z 780.81,A -85,B 0,C 180,E1 10632.786,E2 10632.786} C_VEL
LIN {X 0,Y 545.939,Z 780.81,A -85,B 0,C 180,E1 10637.721,E2 10637.721} C_VEL
LIN {X 0,Y 545.76,Z 780.81,A -85,B 0,C 180,E1 10643.975,E2 10643.975} C_VEL
LIN {X 0,Y 545.581,Z 780.81,A -85,B 0,C 180,E1 10649.896,E2 10649.896} C_VEL
LIN {X 0,Y 545.456,Z 780.81,A -85,B 0,C 180,E1 10655.565,E2 10655.565} C_VEL
LIN {X 0,Y 545.262,Z 780.81,A -85,B 0,C 180,E1 10661.68,E2 10661.68} C_VEL
LIN {X 0,Y 545.308,Z 780.81,A -85,B 0,C 180,E1 10666.682,E2 10666.682} C_VEL
LIN {X 0,Y 549.932,Z 790.766,A -85,B 0,C 180,E1 10667.3,E2 10667.3} C_VEL
LIN {X 0,Y 575.948,Z 839.493,A -85,B 0,C 180,E1 10670.336,E2 10670.336} C_VEL
LIN {X 0,Y 581.648,Z 853.545,A -85,B 0,C 180,E1 10671.084,E2 10671.084} C_VEL
LIN {X 0,Y 578.396,Z 896.238,A -85,B 0,C 180,E1 10672.182,E2 10672.182} C_VEL
LIN {X 0,Y 573.865,Z 940.277,A -85,B 0,C 180,E1 10673.953,E2 10673.953} C_VEL
LIN {X 0,Y 568.335,Z 981.848,A -85,B 0,C 180,E1 10676.301,E2 10676.301} C_VEL
LIN {X 0,Y 563.059,Z 1018.466,A -85,B 0,C 180,E1 10679.056,E2 10679.056} C_VEL
LIN {X 0,Y 557.382,Z 1031.882,A -85,B 0,C 180,E1 10680.067,E2 10680.067} C_VEL
LIN {X 0,Y 552.123,Z 1043.148,A -85,B 0,C 180,E1 10681,E2 10681} C_VEL
LIN {X 0,Y 551.818,Z 1044.666,A -85,B 0,C 180,E1 10681.158,E2 10681.158} C_VEL
LIN {X 0,Y 547.054,Z 1075.841,A -85,B 0,C 180,E1 10684.868,E2 10684.868} C_VEL
LIN {X 0,Y 543.118,Z 1103.985,A -85,B 0,C 180,E1 10689.221,E2 10689.221} C_VEL
LIN {X 0,Y 540.505,Z 1127.491,A -85,B 0,C 180,E1 10694.128,E2 10694.128} C_VEL
LIN {X 0,Y 539.214,Z 1143,A -85,B 0,C 180,E1 10698.706,E2 10698.706} C_VEL
LIN {X 0,Y 538.834,Z 1152.282,A -85,B 0,C 180,E1 10702.749,E2 10702.749} C_VEL
LIN {X 0,Y 538.702,Z 1157.378,A -85,B 0,C 180,E1 10706.783,E2 10706.783} C_VEL
LIN {X 0,Y 538.738,Z 1158.348,A -85,B 0,C 180,E1 10711.606,E2 10711.606} C_VEL
LIN {X 0,Y 538.825,Z 1153.554,A -85,B 0,C 180,E1 10716.44,E2 10716.44} C_VEL
LIN {X 0,Y 539.207,Z 1144.101,A -85,B 0,C 180,E1 10720.903,E2 10720.903} C_VEL
LIN {X 0,Y 540.515,Z 1127.439,A -85,B 0,C 180,E1 10725.875,E2 10725.875} C_VEL
LIN {X 0,Y 543.079,Z 1103.941,A -85,B 0,C 180,E1 10730.778,E2 10730.778} C_VEL
LIN {X 0,Y 547.267,Z 1074.451,A -85,B 0,C 180,E1 10735.339,E2 10735.339} C_VEL
LIN {X 0,Y 552.902,Z 1039.114,A -85,B 0,C 180,E1 10739.468,E2 10739.468} C_VEL
LIN {X 0,Y 559.162,Z 1000.429,A -85,B 0,C 180,E1 10742.888,E2 10742.888} C_VEL
LIN {X 0,Y 565.353,Z 959.226,A -85,B 0,C 180,E1 10745.61,E2 10745.61} C_VEL
LIN {X 0,Y 570.611,Z 917.493,A -85,B 0,C 180,E1 10747.628,E2 10747.628} C_VEL
LIN {X 0,Y 574.913,Z 874.592,A -85,B 0,C 180,E1 10749.052,E2 10749.052} C_VEL
LIN {X 0,Y 575.8,Z 853.744,A -85,B 0,C 180,E1 10749.583,E2 10749.583} C_VEL
LIN {X 0,Y 557.274,Z 816.15,A -85,B 0,C 180,E1 10752.014,E2 10752.014} C_VEL
LIN {X 0,Y 537.712,Z 782.815,A -85,B 0,C 180,E1 10754.606,E2 10754.606} C_VEL
LIN {X 0,Y 537.455,Z 780.81,A -85,B 0,C 180,E1 10754.715,E2 10754.715} C_VEL
LIN {X 0,Y 537.414,Z 780.81,A -85,B 0,C 180,E1 10759.717,E2 10759.717} C_VEL
LIN {X 0,Y 537.474,Z 780.81,A -85,B 0,C 180,E1 10765.795,E2 10765.795} C_VEL
LIN {X 0,Y 537.665,Z 780.81,A -85,B 0,C 180,E1 10771.467,E2 10771.467} C_VEL
LIN {X 0,Y 537.809,Z 780.81,A -85,B 0,C 180,E1 10776.843,E2 10776.843} C_VEL
LIN {X 0,Y 537.949,Z 780.81,A -85,B 0,C 180,E1 10782.755,E2 10782.755} C_VEL
LIN {X 0,Y 538.156,Z 780.81,A -85,B 0,C 180,E1 10788.669,E2 10788.669} C_VEL
LIN {X 0,Y 538.353,Z 780.81,A -85,B 0,C 180,E1 10793.557,E2 10793.557} C_VEL
LIN {X 0,Y 538.515,Z 780.81,A -85,B 0,C 180,E1 10798.395,E2 10798.395} C_VEL
LIN {X 0,Y 538.464,Z 780.81,A -85,B 0,C 180,E1 10803.219,E2 10803.219} C_VEL
LIN {X 0,Y 538.335,Z 780.81,A -85,B 0,C 180,E1 10808.069,E2 10808.069} C_VEL
LIN {X 0,Y 538.138,Z 780.81,A -85,B 0,C 180,E1 10812.982,E2 10812.982} C_VEL
LIN {X 0,Y 537.961,Z 780.81,A -85,B 0,C 180,E1 10817.997,E2 10817.997} C_VEL
LIN {X 0,Y 537.758,Z 780.81,A -85,B 0,C 180,E1 10823.165,E2 10823.165} C_VEL
LIN {X 0,Y 537.646,Z 780.81,A -85,B 0,C 180,E1 10828.539,E2 10828.539} C_VEL
LIN {X 0,Y 537.507,Z 780.81,A -85,B 0,C 180,E1 10834.209,E2 10834.209} C_VEL
LIN {X 0,Y 537.379,Z 780.81,A -85,B 0,C 180,E1 10840.292,E2 10840.292} C_VEL
LIN {X 0,Y 537.525,Z 781.285,A -85,B 0,C 180,E1 10842.806,E2 10842.806} C_VEL
LIN {X 0,Y 540.34,Z 786.858,A -85,B 0,C 180,E1 10843.213,E2 10843.213} C_VEL
LIN {X 0,Y 562.689,Z 827.352,A -85,B 0,C 180,E1 10846.33,E2 10846.33} C_VEL
LIN {X 0,Y 574.448,Z 855.86,A -85,B 0,C 180,E1 10848.33,E2 10848.33} C_VEL
LIN {X 0,Y 570.065,Z 897.95,A -85,B 0,C 180,E1 10849.939,E2 10849.939} C_VEL
LIN {X 0,Y 564.517,Z 939.611,A -85,B 0,C 180,E1 10852.202,E2 10852.202} C_VEL
LIN {X 0,Y 558.168,Z 979.613,A -85,B 0,C 180,E1 10855.159,E2 10855.159} C_VEL
LIN {X 0,Y 551.886,Z 1016.407,A -85,B 0,C 180,E1 10858.79,E2 10858.79} C_VEL
LIN {X 0,Y 546.576,Z 1047.694,A -85,B 0,C 180,E1 10862.861,E2 10862.861} C_VEL
LIN {X 0,Y 542.763,Z 1073.413,A -85,B 0,C 180,E1 10867.277,E2 10867.277} C_VEL
LIN {X 0,Y 540.551,Z 1092.594,A -85,B 0,C 180,E1 10871.669,E2 10871.669} C_VEL
LIN {X 0,Y 539.314,Z 1106.893,A -85,B 0,C 180,E1 10876.223,E2 10876.223} C_VEL
LIN {X 0,Y 538.775,Z 1116.35,A -85,B 0,C 180,E1 10881.127,E2 10881.127} C_VEL
LIN {X 0,Y 538.542,Z 1119.987,A -85,B 0,C 180,E1 10885.172,E2 10885.172} C_VEL
LIN {X 0,Y 538.736,Z 1119.195,A -85,B 0,C 180,E1 10890.001,E2 10890.001} C_VEL
LIN {X 0,Y 538.948,Z 1114.527,A -85,B 0,C 180,E1 10894.02,E2 10894.02} C_VEL
LIN {X 0,Y 539.48,Z 1103.642,A -85,B 0,C 180,E1 10898.863,E2 10898.863} C_VEL
LIN {X 0,Y 540.968,Z 1088.359,A -85,B 0,C 180,E1 10903.325,E2 10903.325} C_VEL
LIN {X 0,Y 543.659,Z 1067.266,A -85,B 0,C 180,E1 10907.804,E2 10907.804} C_VEL
LIN {X 0,Y 547.893,Z 1039.359,A -85,B 0,C 180,E1 10912.216,E2 10912.216} C_VEL
LIN {X 0,Y 553.362,Z 1006.572,A -85,B 0,C 180,E1 10916.126,E2 10916.126} C_VEL
LIN {X 0,Y 559.183,Z 970.463,A -85,B 0,C 180,E1 10919.411,E2 10919.411} C_VEL
LIN {X 0,Y 564.839,Z 932.847,A -85,B 0,C 180,E1 10922.009,E2 10922.009} C_VEL
LIN {X 0,Y 569.754,Z 894.027,A -85,B 0,C 180,E1 10924.026,E2 10924.026} C_VEL
LIN {X 0,Y 572.983,Z 853.779,A -85,B 0,C 180,E1 10925.557,E2 10925.557} C_VEL
LIN {X 0,Y 554.715,Z 813.308,A -85,B 0,C 180,E1 10928.299,E2 10928.299} C_VEL
LIN {X 0,Y 537.517,Z 781.701,A -85,B 0,C 180,E1 10930.492,E2 10930.492} C_VEL
LIN {X 0,Y 537.428,Z 780.81,A -85,B 0,C 180,E1 10930.617,E2 10930.617} C_VEL
LIN {X 0,Y 537.372,Z 780.81,A -85,B 0,C 180,E1 10936.982,E2 10936.982} C_VEL
LIN {X 0,Y 537.443,Z 780.81,A -85,B 0,C 180,E1 10941.932,E2 10941.932} C_VEL
LIN {X 0,Y 537.478,Z 780.81,A -85,B 0,C 180,E1 10947.715,E2 10947.715} C_VEL
LIN {X 0,Y 537.737,Z 780.81,A -85,B 0,C 180,E1 10953.283,E2 10953.283} C_VEL
LIN {X 0,Y 537.841,Z 780.81,A -85,B 0,C 180,E1 10958.579,E2 10958.579} C_VEL
LIN {X 0,Y 537.999,Z 780.81,A -85,B 0,C 180,E1 10963.688,E2 10963.688} C_VEL
LIN {X 0,Y 538.216,Z 780.81,A -85,B 0,C 180,E1 10969.321,E2 10969.321} C_VEL
LIN {X 0,Y 538.456,Z 780.81,A -85,B 0,C 180,E1 10975.169,E2 10975.169} C_VEL
LIN {X 0,Y 538.718,Z 780.81,A -85,B 0,C 180,E1 10979.998,E2 10979.998} C_VEL
LIN {X 0,Y 538.377,Z 780.81,A -85,B 0,C 180,E1 10986.443,E2 10986.443} C_VEL
LIN {X 0,Y 538.184,Z 780.81,A -85,B 0,C 180,E1 10991.331,E2 10991.331} C_VEL
LIN {X 0,Y 538.001,Z 780.81,A -85,B 0,C 180,E1 10997.256,E2 10997.256} C_VEL
LIN {X 0,Y 537.826,Z 780.81,A -85,B 0,C 180,E1 11003.156,E2 11003.156} C_VEL
LIN {X 0,Y 537.649,Z 780.81,A -85,B 0,C 180,E1 11009.391,E2 11009.391} C_VEL
LIN {X 0,Y 537.538,Z 780.81,A -85,B 0,C 180,E1 11015.388,E2 11015.388} C_VEL
LIN {X 0,Y 537.321,Z 780.81,A -85,B 0,C 180,E1 11020.594,E2 11020.594} C_VEL
LIN {X 0,Y 537.38,Z 781.189,A -85,B 0,C 180,E1 11025.945,E2 11025.945} C_VEL
LIN {X 0,Y 542.768,Z 791.713,A -85,B 0,C 180,E1 11026.65,E2 11026.65} C_VEL
LIN {X 0,Y 568.976,Z 841.007,A -85,B 0,C 180,E1 11029.807,E2 11029.807} C_VEL
LIN {X 0,Y 575.268,Z 855.681,A -85,B 0,C 180,E1 11030.647,E2 11030.647} C_VEL
LIN {X 0,Y 571.739,Z 898.823,A -85,B 0,C 180,E1 11031.802,E2 11031.802} C_VEL
LIN {X 0,Y 567.116,Z 941.72,A -85,B 0,C 180,E1 11033.569,E2 11033.569} C_VEL
LIN {X 0,Y 561.328,Z 983.249,A -85,B 0,C 180,E1 11035.964,E2 11035.964} C_VEL
LIN {X 0,Y 555.585,Z 1021.02,A -85,B 0,C 180,E1 11038.883,E2 11038.883} C_VEL
LIN {X 0,Y 551.818,Z 1044.666,A -85,B 0,C 180,E1 11041.158,E2 11041.158} C_VEL
LIN {X 0,Y 546.309,Z 1056.923,A -85,B 0,C 180,E1 11042.337,E2 11042.337} C_VEL
LIN {X 0,Y 540.656,Z 1068.566,A -85,B 0,C 180,E1 11043.585,E2 11043.585} C_VEL
LIN {X 0,Y 536.418,Z 1096.34,A -85,B 0,C 180,E1 11047.647,E2 11047.647} C_VEL
LIN {X 0,Y 533.367,Z 1120.368,A -85,B 0,C 180,E1 11052.267,E2 11052.267} C_VEL
LIN {X 0,Y 531.722,Z 1137.743,A -85,B 0,C 180,E1 11056.858,E2 11056.858} C_VEL
LIN {X 0,Y 531.104,Z 1148.809,A -85,B 0,C 180,E1 11060.996,E2 11060.996} C_VEL
LIN {X 0,Y 530.827,Z 1155.502,A -85,B 0,C 180,E1 11065.1,E2 11065.1} C_VEL
LIN {X 0,Y 530.801,Z 1158.409,A -85,B 0,C 180,E1 11069.999,E2 11069.999} C_VEL
LIN {X 0,Y 530.817,Z 1155.496,A -85,B 0,C 180,E1 11074.898,E2 11074.898} C_VEL
LIN {X 0,Y 531.088,Z 1148.794,A -85,B 0,C 180,E1 11079.002,E2 11079.002} C_VEL
LIN {X 0,Y 531.837,Z 1136.357,A -85,B 0,C 180,E1 11083.556,E2 11083.556} C_VEL
LIN {X 0,Y 533.333,Z 1120.325,A -85,B 0,C 180,E1 11087.732,E2 11087.732} C_VEL
LIN {X 0,Y 536.456,Z 1096.394,A -85,B 0,C 180,E1 11092.35,E2 11092.35} C_VEL
LIN {X 0,Y 540.59,Z 1069.416,A -85,B 0,C 180,E1 11096.342,E2 11096.342} C_VEL
LIN {X 0,Y 546.15,Z 1037.124,A -85,B 0,C 180,E1 11100.067,E2 11100.067} C_VEL
LIN {X 0,Y 552.54,Z 999.337,A -85,B 0,C 180,E1 11103.421,E2 11103.421} C_VEL
LIN {X 0,Y 559.057,Z 958.028,A -85,B 0,C 180,E1 11106.156,E2 11106.156} C_VEL
LIN {X 0,Y 564.513,Z 916.08,A -85,B 0,C 180,E1 11108.182,E2 11108.182} C_VEL
LIN {X 0,Y 568.915,Z 873.068,A -85,B 0,C 180,E1 11109.602,E2 11109.602} C_VEL
LIN {X 0,Y 569.672,Z 856.728,A -85,B 0,C 180,E1 11110.03,E2 11110.03} C_VEL
LIN {X 0,Y 552.084,Z 820.579,A -85,B 0,C 180,E1 11112.439,E2 11112.439} C_VEL
LIN {X 0,Y 531.17,Z 785.597,A -85,B 0,C 180,E1 11115.278,E2 11115.278} C_VEL
LIN {X 0,Y 529.528,Z 780.81,A -85,B 0,C 180,E1 11115.567,E2 11115.567} C_VEL
LIN {X 0,Y 529.465,Z 780.81,A -85,B 0,C 180,E1 11121.117,E2 11121.117} C_VEL
LIN {X 0,Y 529.551,Z 780.81,A -85,B 0,C 180,E1 11127.177,E2 11127.177} C_VEL
LIN {X 0,Y 529.766,Z 780.81,A -85,B 0,C 180,E1 11132.854,E2 11132.854} C_VEL
LIN {X 0,Y 529.906,Z 780.81,A -85,B 0,C 180,E1 11138.247,E2 11138.247} C_VEL
LIN {X 0,Y 530.08,Z 780.81,A -85,B 0,C 180,E1 11143.442,E2 11143.442} C_VEL
LIN {X 0,Y 530.228,Z 780.81,A -85,B 0,C 180,E1 11148.497,E2 11148.497} C_VEL
LIN {X 0,Y 530.453,Z 780.81,A -85,B 0,C 180,E1 11153.461,E2 11153.461} C_VEL
LIN {X 0,Y 530.613,Z 780.81,A -85,B 0,C 180,E1 11158.371,E2 11158.371} C_VEL
LIN {X 0,Y 530.56,Z 780.81,A -85,B 0,C 180,E1 11163.267,E2 11163.267} C_VEL
LIN {X 0,Y 530.416,Z 780.81,A -85,B 0,C 180,E1 11168.19,E2 11168.19} C_VEL
LIN {X 0,Y 530.177,Z 780.81,A -85,B 0,C 180,E1 11174.293,E2 11174.293} C_VEL
LIN {X 0,Y 529.991,Z 780.81,A -85,B 0,C 180,E1 11180.007,E2 11180.007} C_VEL
LIN {X 0,Y 529.776,Z 780.81,A -85,B 0,C 180,E1 11185.329,E2 11185.329} C_VEL
LIN {X 0,Y 529.618,Z 780.81,A -85,B 0,C 180,E1 11191.136,E2 11191.136} C_VEL
LIN {X 0,Y 529.497,Z 780.81,A -85,B 0,C 180,E1 11196.96,E2 11196.96} C_VEL
LIN {X 0,Y 529.553,Z 781.196,A -85,B 0,C 180,E1 11201.916,E2 11201.916} C_VEL
LIN {X 0,Y 532.105,Z 786.558,A -85,B 0,C 180,E1 11202.307,E2 11202.307} C_VEL
LIN {X 0,Y 554.237,Z 825.547,A -85,B 0,C 180,E1 11205.484,E2 11205.484} C_VEL
LIN {X 0,Y 568.11,Z 858.168,A -85,B 0,C 180,E1 11207.874,E2 11207.874} C_VEL
LIN {X 0,Y 563.455,Z 900.836,A -85,B 0,C 180,E1 11209.561,E2 11209.561} C_VEL
LIN {X 0,Y 557.934,Z 940.384,A -85,B 0,C 180,E1 11211.752,E2 11211.752} C_VEL
LIN {X 0,Y 551.442,Z 979.8,A -85,B 0,C 180,E1 11214.699,E2 11214.699} C_VEL
LIN {X 0,Y 545.055,Z 1015.232,A -85,B 0,C 180,E1 11218.215,E2 11218.215} C_VEL
LIN {X 0,Y 539.626,Z 1045.55,A -85,B 0,C 180,E1 11222.143,E2 11222.143} C_VEL
LIN {X 0,Y 535.819,Z 1069.958,A -85,B 0,C 180,E1 11226.246,E2 11226.246} C_VEL
LIN {X 0,Y 532.908,Z 1091.198,A -85,B 0,C 180,E1 11230.969,E2 11230.969} C_VEL
LIN {X 0,Y 531.468,Z 1107.054,A -85,B 0,C 180,E1 11236.015,E2 11236.015} C_VEL
LIN {X 0,Y 530.913,Z 1116.566,A -85,B 0,C 180,E1 11240.995,E2 11240.995} C_VEL
LIN {X 0,Y 530.649,Z 1120.293,A -85,B 0,C 180,E1 11245.24,E2 11245.24} C_VEL
LIN {X 0,Y 530.84,Z 1119.504,A -85,B 0,C 180,E1 11250.001,E2 11250.001} C_VEL
LIN {X 0,Y 531.088,Z 1114.872,A -85,B 0,C 180,E1 11254.08,E2 11254.08} C_VEL
LIN {X 0,Y 531.647,Z 1104.049,A -85,B 0,C 180,E1 11258.995,E2 11258.995} C_VEL
LIN {X 0,Y 533.208,Z 1088.831,A -85,B 0,C 180,E1 11263.522,E2 11263.522} C_VEL
LIN {X 0,Y 536.043,Z 1067.781,A -85,B 0,C 180,E1 11268.066,E2 11268.066} C_VEL
LIN {X 0,Y 540.578,Z 1039.469,A -85,B 0,C 180,E1 11272.597,E2 11272.597} C_VEL
LIN {X 0,Y 546.546,Z 1005.277,A -85,B 0,C 180,E1 11276.699,E2 11276.699} C_VEL
LIN {X 0,Y 553.023,Z 966.82,A -85,B 0,C 180,E1 11280.166,E2 11280.166} C_VEL
LIN {X 0,Y 559.45,Z 924.329,A -85,B 0,C 180,E1 11282.997,E2 11282.997} C_VEL
LIN {X 0,Y 564.704,Z 882.34,A -85,B 0,C 180,E1 11284.997,E2 11284.997} C_VEL
LIN {X 0,Y 566.519,Z 856.608,A -85,B 0,C 180,E1 11285.967,E2 11285.967} C_VEL
LIN {X 0,Y 548.625,Z 816.49,A -85,B 0,C 180,E1 11288.764,E2 11288.764} C_VEL
LIN {X 0,Y 529.492,Z 781.647,A -85,B 0,C 180,E1 11291.296,E2 11291.296} C_VEL
LIN {X 0,Y 529.466,Z 780.81,A -85,B 0,C 180,E1 11292.101,E2 11292.101} C_VEL
LIN {X 0,Y 529.427,Z 780.81,A -85,B 0,C 180,E1 11297.912,E2 11297.912} C_VEL
LIN {X 0,Y 529.475,Z 780.81,A -85,B 0,C 180,E1 11303.182,E2 11303.182} C_VEL
LIN {X 0,Y 529.603,Z 780.81,A -85,B 0,C 180,E1 11309.1,E2 11309.1} C_VEL
LIN {X 0,Y 529.818,Z 780.81,A -85,B 0,C 180,E1 11314.673,E2 11314.673} C_VEL
LIN {X 0,Y 530.033,Z 780.81,A -85,B 0,C 180,E1 11320.192,E2 11320.192} C_VEL
LIN {X 0,Y 530.122,Z 780.81,A -85,B 0,C 180,E1 11325.738,E2 11325.738} C_VEL
LIN {X 0,Y 530.433,Z 780.81,A -85,B 0,C 180,E1 11331.81,E2 11331.81} C_VEL
LIN {X 0,Y 530.664,Z 780.81,A -85,B 0,C 180,E1 11336.733,E2 11336.733} C_VEL
LIN {X 0,Y 530.732,Z 780.81,A -85,B 0,C 180,E1 11341.629,E2 11341.629} C_VEL
LIN {X 0,Y 530.475,Z 780.81,A -85,B 0,C 180,E1 11346.539,E2 11346.539} C_VEL
LIN {X 0,Y 530.258,Z 780.81,A -85,B 0,C 180,E1 11351.502,E2 11351.502} C_VEL
LIN {X 0,Y 530.142,Z 780.81,A -85,B 0,C 180,E1 11356.556,E2 11356.556} C_VEL
LIN {X 0,Y 529.931,Z 780.81,A -85,B 0,C 180,E1 11361.752,E2 11361.752} C_VEL
LIN {X 0,Y 529.754,Z 780.81,A -85,B 0,C 180,E1 11367.837,E2 11367.837} C_VEL
LIN {X 0,Y 529.671,Z 780.81,A -85,B 0,C 180,E1 11374.171,E2 11374.171} C_VEL
LIN {X 0,Y 529.419,Z 780.81,A -85,B 0,C 180,E1 11379.586,E2 11379.586} C_VEL
LIN {X 0,Y 529.419,Z 780.81,A -85,B 0,C 180,E1 11385.131,E2 11385.131} C_VEL
LIN {X 0,Y 531.884,Z 786.532,A -85,B 0,C 180,E1 11385.495,E2 11385.495} C_VEL
LIN {X 0,Y 557.348,Z 832.892,A -85,B 0,C 180,E1 11388.681,E2 11388.681} C_VEL
LIN {X 0,Y 568.82,Z 857.246,A -85,B 0,C 180,E1 11390.178,E2 11390.178} C_VEL
LIN {X 0,Y 565.191,Z 900.709,A -85,B 0,C 180,E1 11391.391,E2 11391.391} C_VEL
LIN {X 0,Y 560.43,Z 942.618,A -85,B 0,C 180,E1 11393.154,E2 11393.154} C_VEL
LIN {X 0,Y 554.361,Z 984.415,A -85,B 0,C 180,E1 11395.604,E2 11395.604} C_VEL
LIN {X 0,Y 548.143,Z 1023.43,A -85,B 0,C 180,E1 11398.695,E2 11398.695} C_VEL
LIN {X 0,Y 542.536,Z 1057.216,A -85,B 0,C 180,E1 11402.19,E2 11402.19} C_VEL
LIN {X 0,Y 540.656,Z 1068.566,A -85,B 0,C 180,E1 11403.585,E2 11403.585} C_VEL
LIN {X 0,Y 535.119,Z 1079.607,A -85,B 0,C 180,E1 11404.918,E2 11404.918} C_VEL
LIN {X 0,Y 529.751,Z 1089.964,A -85,B 0,C 180,E1 11406.326,E2 11406.326} C_VEL
LIN {X 0,Y 526.384,Z 1114.112,A -85,B 0,C 180,E1 11410.715,E2 11410.715} C_VEL
LIN {X 0,Y 524.25,Z 1133.358,A -85,B 0,C 180,E1 11415.391,E2 11415.391} C_VEL
LIN {X 0,Y 523.277,Z 1146.591,A -85,B 0,C 180,E1 11420.021,E2 11420.021} C_VEL
LIN {X 0,Y 522.988,Z 1154.23,A -85,B 0,C 180,E1 11424.195,E2 11424.195} C_VEL
LIN {X 0,Y 522.952,Z 1157.788,A -85,B 0,C 180,E1 11428.343,E2 11428.343} C_VEL
LIN {X 0,Y 522.937,Z 1157.784,A -85,B 0,C 180,E1 11431.655,E2 11431.655} C_VEL
LIN {X 0,Y 523.051,Z 1152.985,A -85,B 0,C 180,E1 11436.635,E2 11436.635} C_VEL
LIN {X 0,Y 523.449,Z 1143.912,A -85,B 0,C 180,E1 11441.095,E2 11441.095} C_VEL
LIN {X 0,Y 524.842,Z 1127.812,A -85,B 0,C 180,E1 11446.105,E2 11446.105} C_VEL
LIN {X 0,Y 527.461,Z 1106.082,A -85,B 0,C 180,E1 11450.894,E2 11450.894} C_VEL
LIN {X 0,Y 531.506,Z 1079.915,A -85,B 0,C 180,E1 11455.242,E2 11455.242} C_VEL
LIN {X 0,Y 536.807,Z 1049.565,A -85,B 0,C 180,E1 11459.147,E2 11459.147} C_VEL
LIN {X 0,Y 543.463,Z 1012.229,A -85,B 0,C 180,E1 11462.832,E2 11462.832} C_VEL
LIN {X 0,Y 550.612,Z 970.354,A -85,B 0,C 180,E1 11465.915,E2 11465.915} C_VEL
LIN {X 0,Y 557.06,Z 926.006,A -85,B 0,C 180,E1 11468.277,E2 11468.277} C_VEL
LIN {X 0,Y 562.29,Z 879.725,A -85,B 0,C 180,E1 11469.942,E2 11469.942} C_VEL
LIN {X 0,Y 563.561,Z 859.574,A -85,B 0,C 180,E1 11470.494,E2 11470.494} C_VEL
LIN {X 0,Y 546.052,Z 823.252,A -85,B 0,C 180,E1 11472.992,E2 11472.992} C_VEL
LIN {X 0,Y 524.103,Z 786.569,A -85,B 0,C 180,E1 11476.072,E2 11476.072} C_VEL
LIN {X 0,Y 521.613,Z 780.81,A -85,B 0,C 180,E1 11476.545,E2 11476.545} C_VEL
LIN {X 0,Y 521.54,Z 780.81,A -85,B 0,C 180,E1 11482.533,E2 11482.533} C_VEL
LIN {X 0,Y 521.667,Z 780.81,A -85,B 0,C 180,E1 11488.583,E2 11488.583} C_VEL
LIN {X 0,Y 521.861,Z 780.81,A -85,B 0,C 180,E1 11494.264,E2 11494.264} C_VEL
LIN {X 0,Y 522.035,Z 780.81,A -85,B 0,C 180,E1 11499.681,E2 11499.681} C_VEL
LIN {X 0,Y 522.192,Z 780.81,A -85,B 0,C 180,E1 11504.909,E2 11504.909} C_VEL
LIN {X 0,Y 522.409,Z 780.81,A -85,B 0,C 180,E1 11510.01,E2 11510.01} C_VEL
LIN {X 0,Y 522.626,Z 780.81,A -85,B 0,C 180,E1 11515.027,E2 11515.027} C_VEL
LIN {X 0,Y 522.896,Z 780.81,A -85,B 0,C 180,E1 11520.003,E2 11520.003} C_VEL
LIN {X 0,Y 522.598,Z 780.81,A -85,B 0,C 180,E1 11526.643,E2 11526.643} C_VEL
LIN {X 0,Y 522.35,Z 780.81,A -85,B 0,C 180,E1 11531.684,E2 11531.684} C_VEL
LIN {X 0,Y 522.155,Z 780.81,A -85,B 0,C 180,E1 11537.255,E2 11537.255} C_VEL
LIN {X 0,Y 521.953,Z 780.81,A -85,B 0,C 180,E1 11542.117,E2 11542.117} C_VEL
LIN {X 0,Y 521.842,Z 780.81,A -85,B 0,C 180,E1 11547.599,E2 11547.599} C_VEL
LIN {X 0,Y 521.689,Z 780.81,A -85,B 0,C 180,E1 11553.387,E2 11553.387} C_VEL
LIN {X 0,Y 521.57,Z 780.81,A -85,B 0,C 180,E1 11559.593,E2 11559.593} C_VEL
LIN {X 0,Y 521.577,Z 780.851,A -85,B 0,C 180,E1 11560.976,E2 11560.976} C_VEL
LIN {X 0,Y 523.966,Z 786.475,A -85,B 0,C 180,E1 11561.371,E2 11561.371} C_VEL
LIN {X 0,Y 545.619,Z 823.409,A -85,B 0,C 180,E1 11564.573,E2 11564.573} C_VEL
LIN {X 0,Y 560.84,Z 858.192,A -85,B 0,C 180,E1 11567.232,E2 11567.232} C_VEL
LIN {X 0,Y 561.804,Z 862.508,A -85,B 0,C 180,E1 11567.488,E2 11567.488} C_VEL
LIN {X 0,Y 556.176,Z 909.43,A -85,B 0,C 180,E1 11569.453,E2 11569.453} C_VEL
LIN {X 0,Y 549.583,Z 952.317,A -85,B 0,C 180,E1 11572.049,E2 11572.049} C_VEL
LIN {X 0,Y 543.026,Z 988.997,A -85,B 0,C 180,E1 11575.046,E2 11575.046} C_VEL
LIN {X 0,Y 537.085,Z 1020.686,A -85,B 0,C 180,E1 11578.399,E2 11578.399} C_VEL
LIN {X 0,Y 531.354,Z 1051.239,A -85,B 0,C 180,E1 11582.586,E2 11582.586} C_VEL
LIN {X 0,Y 527.127,Z 1076.789,A -85,B 0,C 180,E1 11587.233,E2 11587.233} C_VEL
LIN {X 0,Y 524.7,Z 1096.62,A -85,B 0,C 180,E1 11592.177,E2 11592.177} C_VEL
LIN {X 0,Y 523.471,Z 1109.167,A -85,B 0,C 180,E1 11596.649,E2 11596.649} C_VEL
LIN {X 0,Y 523.023,Z 1116.783,A -85,B 0,C 180,E1 11600.858,E2 11600.858} C_VEL
LIN {X 0,Y 522.763,Z 1120.504,A -85,B 0,C 180,E1 11605.026,E2 11605.026} C_VEL
LIN {X 0,Y 522.945,Z 1119.813,A -85,B 0,C 180,E1 11610.001,E2 11610.001} C_VEL
LIN {X 0,Y 523.225,Z 1115.218,A -85,B 0,C 180,E1 11614.141,E2 11614.141} C_VEL
LIN {X 0,Y 523.814,Z 1104.455,A -85,B 0,C 180,E1 11619.13,E2 11619.13} C_VEL
LIN {X 0,Y 525.456,Z 1089.287,A -85,B 0,C 180,E1 11623.725,E2 11623.725} C_VEL
LIN {X 0,Y 528.463,Z 1068.27,A -85,B 0,C 180,E1 11628.334,E2 11628.334} C_VEL
LIN {X 0,Y 533.231,Z 1039.997,A -85,B 0,C 180,E1 11632.926,E2 11632.926} C_VEL
LIN {X 0,Y 539.097,Z 1007.747,A -85,B 0,C 180,E1 11636.872,E2 11636.872} C_VEL
LIN {X 0,Y 545.174,Z 973.291,A -85,B 0,C 180,E1 11640.105,E2 11640.105} C_VEL
LIN {X 0,Y 551.323,Z 936.077,A -85,B 0,C 180,E1 11642.775,E2 11642.775} C_VEL
LIN {X 0,Y 556.941,Z 894.845,A -85,B 0,C 180,E1 11644.976,E2 11644.976} C_VEL
LIN {X 0,Y 560.255,Z 859.845,A -85,B 0,C 180,E1 11646.356,E2 11646.356} C_VEL
LIN {X 0,Y 542.543,Z 819.784,A -85,B 0,C 180,E1 11649.236,E2 11649.236} C_VEL
LIN {X 0,Y 521.734,Z 782.293,A -85,B 0,C 180,E1 11652.093,E2 11652.093} C_VEL
LIN {X 0,Y 521.557,Z 780.81,A -85,B 0,C 180,E1 11652.296,E2 11652.296} C_VEL
LIN {X 0,Y 521.526,Z 780.81,A -85,B 0,C 180,E1 11658.214,E2 11658.214} C_VEL
LIN {X 0,Y 521.52,Z 780.81,A -85,B 0,C 180,E1 11664.225,E2 11664.225} C_VEL
LIN {X 0,Y 521.745,Z 780.81,A -85,B 0,C 180,E1 11670.33,E2 11670.33} C_VEL
LIN {X 0,Y 521.908,Z 780.81,A -85,B 0,C 180,E1 11676.089,E2 11676.089} C_VEL
LIN {X 0,Y 522.102,Z 780.81,A -85,B 0,C 180,E1 11681.436,E2 11681.436} C_VEL
LIN {X 0,Y 522.247,Z 780.81,A -85,B 0,C 180,E1 11686.616,E2 11686.616} C_VEL
LIN {X 0,Y 522.513,Z 780.81,A -85,B 0,C 180,E1 11691.685,E2 11691.685} C_VEL
LIN {X 0,Y 522.773,Z 780.81,A -85,B 0,C 180,E1 11696.684,E2 11696.684} C_VEL
LIN {X 0,Y 522.839,Z 780.81,A -85,B 0,C 180,E1 11701.653,E2 11701.653} C_VEL
LIN {X 0,Y 522.559,Z 780.81,A -85,B 0,C 180,E1 11706.639,E2 11706.639} C_VEL
LIN {X 0,Y 522.349,Z 780.81,A -85,B 0,C 180,E1 11711.679,E2 11711.679} C_VEL
LIN {X 0,Y 522.161,Z 780.81,A -85,B 0,C 180,E1 11717.251,E2 11717.251} C_VEL
LIN {X 0,Y 521.991,Z 780.81,A -85,B 0,C 180,E1 11722.123,E2 11722.123} C_VEL
LIN {X 0,Y 521.877,Z 780.81,A -85,B 0,C 180,E1 11727.591,E2 11727.591} C_VEL
LIN {X 0,Y 521.728,Z 780.81,A -85,B 0,C 180,E1 11733.379,E2 11733.379} C_VEL
LIN {X 0,Y 521.543,Z 780.81,A -85,B 0,C 180,E1 11739.588,E2 11739.588} C_VEL
LIN {X 0,Y 521.526,Z 781.232,A -85,B 0,C 180,E1 11744.324,E2 11744.324} C_VEL
LIN {X 0,Y 526.564,Z 791.231,A -85,B 0,C 180,E1 11745.039,E2 11745.039} C_VEL
LIN {X 0,Y 550.515,Z 834.358,A -85,B 0,C 180,E1 11748.114,E2 11748.114} C_VEL
LIN {X 0,Y 562.461,Z 859.828,A -85,B 0,C 180,E1 11749.728,E2 11749.728} C_VEL
LIN {X 0,Y 558.341,Z 905.388,A -85,B 0,C 180,E1 11751.066,E2 11751.066} C_VEL
LIN {X 0,Y 553.415,Z 945.932,A -85,B 0,C 180,E1 11752.857,E2 11752.857} C_VEL
LIN {X 0,Y 547.292,Z 986.28,A -85,B 0,C 180,E1 11755.286,E2 11755.286} C_VEL
LIN {X 0,Y 540.648,Z 1026.441,A -85,B 0,C 180,E1 11758.56,E2 11758.56} C_VEL
LIN {X 0,Y 534.393,Z 1062.156,A -85,B 0,C 180,E1 11762.416,E2 11762.416} C_VEL
LIN {X 0,Y 529.751,Z 1089.964,A -85,B 0,C 180,E1 11766.326,E2 11766.326} C_VEL
LIN {X 0,Y 524.415,Z 1099.671,A -85,B 0,C 180,E1 11767.81,E2 11767.81} C_VEL
LIN {X 0,Y 519.41,Z 1108.653,A -85,B 0,C 180,E1 11769.368,E2 11769.368} C_VEL
LIN {X 0,Y 516.954,Z 1128.37,A -85,B 0,C 180,E1 11773.876,E2 11773.876} C_VEL
LIN {X 0,Y 515.533,Z 1143.707,A -85,B 0,C 180,E1 11778.752,E2 11778.752} C_VEL
LIN {X 0,Y 515.142,Z 1152.715,A -85,B 0,C 180,E1 11783.261,E2 11783.261} C_VEL
LIN {X 0,Y 515.026,Z 1156.536,A -85,B 0,C 180,E1 11786.635,E2 11786.635} C_VEL
LIN {X 0,Y 515.036,Z 1157.503,A -85,B 0,C 180,E1 11791.68,E2 11791.68} C_VEL
LIN {X 0,Y 515.112,Z 1153.937,A -85,B 0,C 180,E1 11795.892,E2 11795.892} C_VEL
LIN {X 0,Y 515.522,Z 1144.975,A -85,B 0,C 180,E1 11800.698,E2 11800.698} C_VEL
LIN {X 0,Y 516.639,Z 1131.512,A -85,B 0,C 180,E1 11805.261,E2 11805.261} C_VEL
LIN {X 0,Y 519.19,Z 1110.897,A -85,B 0,C 180,E1 11810.219,E2 11810.219} C_VEL
LIN {X 0,Y 523.331,Z 1084.48,A -85,B 0,C 180,E1 11814.915,E2 11814.915} C_VEL
LIN {X 0,Y 529.134,Z 1052.409,A -85,B 0,C 180,E1 11819.227,E2 11819.227} C_VEL
LIN {X 0,Y 535.764,Z 1016.793,A -85,B 0,C 180,E1 11822.883,E2 11822.883} C_VEL
LIN {X 0,Y 542.488,Z 979.535,A -85,B 0,C 180,E1 11825.799,E2 11825.799} C_VEL
LIN {X 0,Y 549.049,Z 938.945,A -85,B 0,C 180,E1 11828.178,E2 11828.178} C_VEL
LIN {X 0,Y 554.87,Z 894.238,A -85,B 0,C 180,E1 11830.019,E2 11830.019} C_VEL
LIN {X 0,Y 557.399,Z 862.254,A -85,B 0,C 180,E1 11830.966,E2 11830.966} C_VEL
LIN {X 0,Y 540.055,Z 826.125,A -85,B 0,C 180,E1 11833.556,E2 11833.556} C_VEL
LIN {X 0,Y 518.892,Z 791.119,A -85,B 0,C 180,E1 11836.603,E2 11836.603} C_VEL
LIN {X 0,Y 513.918,Z 782.71,A -85,B 0,C 180,E1 11837.387,E2 11837.387} C_VEL
LIN {X 0,Y 513.68,Z 780.81,A -85,B 0,C 180,E1 11837.525,E2 11837.525} C_VEL
LIN {X 0,Y 513.636,Z 780.81,A -85,B 0,C 180,E1 11843.967,E2 11843.967} C_VEL
LIN {X 0,Y 513.791,Z 780.81,A -85,B 0,C 180,E1 11850.01,E2 11850.01} C_VEL
LIN {X 0,Y 513.965,Z 780.81,A -85,B 0,C 180,E1 11855.701,E2 11855.701} C_VEL
LIN {X 0,Y 514.141,Z 780.81,A -85,B 0,C 180,E1 11861.143,E2 11861.143} C_VEL
LIN {X 0,Y 514.305,Z 780.81,A -85,B 0,C 180,E1 11866.41,E2 11866.41} C_VEL
LIN {X 0,Y 514.588,Z 780.81,A -85,B 0,C 180,E1 11871.561,E2 11871.561} C_VEL
LIN {X 0,Y 514.852,Z 780.81,A -85,B 0,C 180,E1 11876.638,E2 11876.638} C_VEL
LIN {X 0,Y 514.919,Z 780.81,A -85,B 0,C 180,E1 11881.684,E2 11881.684} C_VEL
LIN {X 0,Y 514.706,Z 780.81,A -85,B 0,C 180,E1 11886.745,E2 11886.745} C_VEL
LIN {X 0,Y 514.423,Z 780.81,A -85,B 0,C 180,E1 11891.867,E2 11891.867} C_VEL
LIN {X 0,Y 514.274,Z 780.81,A -85,B 0,C 180,E1 11897.087,E2 11897.087} C_VEL
LIN {X 0,Y 514.025,Z 780.81,A -85,B 0,C 180,E1 11902.467,E2 11902.467} C_VEL
LIN {X 0,Y 513.889,Z 780.81,A -85,B 0,C 180,E1 11908.098,E2 11908.098} C_VEL
LIN {X 0,Y 513.696,Z 780.81,A -85,B 0,C 180,E1 11913.977,E2 11913.977} C_VEL
LIN {X 0,Y 513.64,Z 780.81,A -85,B 0,C 180,E1 11919.993,E2 11919.993} C_VEL
LIN {X 0,Y 515.993,Z 786.405,A -85,B 0,C 180,E1 11920.408,E2 11920.408} C_VEL
LIN {X 0,Y 536.822,Z 821.214,A -85,B 0,C 180,E1 11923.597,E2 11923.597} C_VEL
LIN {X 0,Y 552.919,Z 856.402,A -85,B 0,C 180,E1 11926.431,E2 11926.431} C_VEL
LIN {X 0,Y 555.582,Z 864.79,A -85,B 0,C 180,E1 11927.028,E2 11927.028} C_VEL
LIN {X 0,Y 549.887,Z 910.301,A -85,B 0,C 180,E1 11928.966,E2 11928.966} C_VEL
LIN {X 0,Y 543.103,Z 952.734,A -85,B 0,C 180,E1 11931.562,E2 11931.562} C_VEL
LIN {X 0,Y 535.904,Z 991.244,A -85,B 0,C 180,E1 11934.76,E2 11934.76} C_VEL
LIN {X 0,Y 529.386,Z 1024.201,A -85,B 0,C 180,E1 11938.366,E2 11938.366} C_VEL
LIN {X 0,Y 524.031,Z 1051.533,A -85,B 0,C 180,E1 11942.209,E2 11942.209} C_VEL
LIN {X 0,Y 519.582,Z 1077.108,A -85,B 0,C 180,E1 11946.93,E2 11946.93} C_VEL
LIN {X 0,Y 516.933,Z 1097.119,A -85,B 0,C 180,E1 11952.004,E2 11952.004} C_VEL
LIN {X 0,Y 515.625,Z 1109.352,A -85,B 0,C 180,E1 11956.442,E2 11956.442} C_VEL
LIN {X 0,Y 515.14,Z 1117.001,A -85,B 0,C 180,E1 11960.717,E2 11960.717} C_VEL
LIN {X 0,Y 514.879,Z 1120.757,A -85,B 0,C 180,E1 11964.95,E2 11964.95} C_VEL
LIN {X 0,Y 515.049,Z 1120.122,A -85,B 0,C 180,E1 11970.001,E2 11970.001} C_VEL
LIN {X 0,Y 515.327,Z 1114.147,A -85,B 0,C 180,E1 11975.048,E2 11975.048} C_VEL
LIN {X 0,Y 516.236,Z 1102.558,A -85,B 0,C 180,E1 11980.116,E2 11980.116} C_VEL
LIN {X 0,Y 518.436,Z 1084.673,A -85,B 0,C 180,E1 11985.209,E2 11985.209} C_VEL
LIN {X 0,Y 522.164,Z 1061.047,A -85,B 0,C 180,E1 11990.014,E2 11990.014} C_VEL
LIN {X 0,Y 527.327,Z 1032.721,A -85,B 0,C 180,E1 11994.327,E2 11994.327} C_VEL
LIN {X 0,Y 533.345,Z 1001.367,A -85,B 0,C 180,E1 11997.987,E2 11997.987} C_VEL
LIN {X 0,Y 539.714,Z 966.366,A -85,B 0,C 180,E1 12001.15,E2 12001.15} C_VEL
LIN {X 0,Y 546.594,Z 924.124,A -85,B 0,C 180,E1 12003.999,E2 12003.999} C_VEL
LIN {X 0,Y 552.482,Z 879.499,A -85,B 0,C 180,E1 12006.132,E2 12006.132} C_VEL
LIN {X 0,Y 553.984,Z 862.948,A -85,B 0,C 180,E1 12006.759,E2 12006.759} C_VEL
LIN {X 0,Y 536.787,Z 823.577,A -85,B 0,C 180,E1 12009.676,E2 12009.676} C_VEL
LIN {X 0,Y 515.72,Z 786.135,A -85,B 0,C 180,E1 12012.672,E2 12012.672} C_VEL
LIN {X 0,Y 513.667,Z 780.81,A -85,B 0,C 180,E1 12013.016,E2 12013.016} C_VEL
LIN {X 0,Y 513.647,Z 780.81,A -85,B 0,C 180,E1 12019.899,E2 12019.899} C_VEL
LIN {X 0,Y 513.639,Z 780.81,A -85,B 0,C 180,E1 12026.019,E2 12026.019} C_VEL
LIN {X 0,Y 513.889,Z 780.81,A -85,B 0,C 180,E1 12031.937,E2 12031.937} C_VEL
LIN {X 0,Y 514.045,Z 780.81,A -85,B 0,C 180,E1 12037.534,E2 12037.534} C_VEL
LIN {X 0,Y 514.249,Z 780.81,A -85,B 0,C 180,E1 12042.912,E2 12042.912} C_VEL
LIN {X 0,Y 514.409,Z 780.81,A -85,B 0,C 180,E1 12048.133,E2 12048.133} C_VEL
LIN {X 0,Y 514.662,Z 780.81,A -85,B 0,C 180,E1 12053.254,E2 12053.254} C_VEL
LIN {X 0,Y 514.871,Z 780.81,A -85,B 0,C 180,E1 12058.316,E2 12058.316} C_VEL
LIN {X 0,Y 514.749,Z 780.81,A -85,B 0,C 180,E1 12063.509,E2 12063.509} C_VEL
LIN {X 0,Y 514.598,Z 780.81,A -85,B 0,C 180,E1 12068.439,E2 12068.439} C_VEL
LIN {X 0,Y 514.334,Z 780.81,A -85,B 0,C 180,E1 12074.175,E2 12074.175} C_VEL
LIN {X 0,Y 514.165,Z 780.81,A -85,B 0,C 180,E1 12079.868,E2 12079.868} C_VEL
LIN {X 0,Y 513.975,Z 780.81,A -85,B 0,C 180,E1 12086.16,E2 12086.16} C_VEL
LIN {X 0,Y 513.825,Z 780.81,A -85,B 0,C 180,E1 12091.953,E2 12091.953} C_VEL
LIN {X 0,Y 513.647,Z 780.81,A -85,B 0,C 180,E1 12098.145,E2 12098.145} C_VEL
LIN {X 0,Y 513.579,Z 780.81,A -85,B 0,C 180,E1 12103.434,E2 12103.434} C_VEL
LIN {X 0,Y 516.192,Z 786.673,A -85,B 0,C 180,E1 12103.85,E2 12103.85} C_VEL
LIN {X 0,Y 541.996,Z 832.521,A -85,B 0,C 180,E1 12107.304,E2 12107.304} C_VEL
LIN {X 0,Y 556.185,Z 862.911,A -85,B 0,C 180,E1 12109.302,E2 12109.302} C_VEL
LIN {X 0,Y 551.622,Z 909.162,A -85,B 0,C 180,E1 12110.703,E2 12110.703} C_VEL
LIN {X 0,Y 545.668,Z 953.899,A -85,B 0,C 180,E1 12112.794,E2 12112.794} C_VEL
LIN {X 0,Y 539.423,Z 992.822,A -85,B 0,C 180,E1 12115.317,E2 12115.317} C_VEL
LIN {X 0,Y 533.274,Z 1028.123,A -85,B 0,C 180,E1 12118.311,E2 12118.311} C_VEL
LIN {X 0,Y 527.151,Z 1061.75,A -85,B 0,C 180,E1 12122.004,E2 12122.004} C_VEL
LIN {X 0,Y 521.917,Z 1091.767,A -85,B 0,C 180,E1 12126.313,E2 12126.313} C_VEL
LIN {X 0,Y 519.41,Z 1108.653,A -85,B 0,C 180,E1 12129.368,E2 12129.368} C_VEL
LIN {X 0,Y 517.685,Z 1112.901,A -85,B 0,C 180,E1 12130.193,E2 12130.193} C_VEL
LIN {X 0,Y 509.721,Z 1123.552,A -85,B 0,C 180,E1 12132.458,E2 12132.458} C_VEL
LIN {X 0,Y 509.533,Z 1124.459,A -85,B 0,C 180,E1 12132.682,E2 12132.682} C_VEL
LIN {X 0,Y 507.986,Z 1139.44,A -85,B 0,C 180,E1 12137.108,E2 12137.108} C_VEL
LIN {X 0,Y 507.315,Z 1151.15,A -85,B 0,C 180,E1 12142.296,E2 12142.296} C_VEL
LIN {X 0,Y 507.136,Z 1156.255,A -85,B 0,C 180,E1 12146.583,E2 12146.583} C_VEL
LIN {X 0,Y 507.138,Z 1157.567,A -85,B 0,C 180,E1 12149.999,E2 12149.999} C_VEL
LIN {X 0,Y 507.165,Z 1154.649,A -85,B 0,C 180,E1 12155.127,E2 12155.127} C_VEL
LIN {X 0,Y 507.43,Z 1147.945,A -85,B 0,C 180,E1 12159.426,E2 12159.426} C_VEL
LIN {X 0,Y 508.452,Z 1134.508,A -85,B 0,C 180,E1 12164.523,E2 12164.523} C_VEL
LIN {X 0,Y 510.464,Z 1117.637,A -85,B 0,C 180,E1 12169.003,E2 12169.003} C_VEL
LIN {X 0,Y 514.334,Z 1093.27,A -85,B 0,C 180,E1 12173.826,E2 12173.826} C_VEL
LIN {X 0,Y 520.12,Z 1062.411,A -85,B 0,C 180,E1 12178.407,E2 12178.407} C_VEL
LIN {X 0,Y 527.098,Z 1026.35,A -85,B 0,C 180,E1 12182.461,E2 12182.461} C_VEL
LIN {X 0,Y 534.674,Z 986.93,A -85,B 0,C 180,E1 12185.779,E2 12185.779} C_VEL
LIN {X 0,Y 541.575,Z 946.792,A -85,B 0,C 180,E1 12188.286,E2 12188.286} C_VEL
LIN {X 0,Y 547.444,Z 905.823,A -85,B 0,C 180,E1 12190.143,E2 12190.143} C_VEL
LIN {X 0,Y 551.213,Z 864.958,A -85,B 0,C 180,E1 12191.449,E2 12191.449} C_VEL
LIN {X 0,Y 534.076,Z 828.892,A -85,B 0,C 180,E1 12194.128,E2 12194.128} C_VEL
LIN {X 0,Y 511.796,Z 792.105,A -85,B 0,C 180,E1 12197.461,E2 12197.461} C_VEL
LIN {X 0,Y 506.005,Z 782.759,A -85,B 0,C 180,E1 12198.407,E2 12198.407} C_VEL
LIN {X 0,Y 505.764,Z 780.81,A -85,B 0,C 180,E1 12198.65,E2 12198.65} C_VEL
LIN {X 0,Y 505.75,Z 780.81,A -85,B 0,C 180,E1 12205.421,E2 12205.421} C_VEL
LIN {X 0,Y 505.931,Z 780.81,A -85,B 0,C 180,E1 12211.461,E2 12211.461} C_VEL
LIN {X 0,Y 506.159,Z 780.81,A -85,B 0,C 180,E1 12217.739,E2 12217.739} C_VEL
LIN {X 0,Y 506.323,Z 780.81,A -85,B 0,C 180,E1 12222.748,E2 12222.748} C_VEL
LIN {X 0,Y 506.468,Z 780.81,A -85,B 0,C 180,E1 12227.95,E2 12227.95} C_VEL
LIN {X 0,Y 506.719,Z 780.81,A -85,B 0,C 180,E1 12233.153,E2 12233.153} C_VEL
LIN {X 0,Y 506.924,Z 780.81,A -85,B 0,C 180,E1 12238.295,E2 12238.295} C_VEL
LIN {X 0,Y 506.88,Z 780.81,A -85,B 0,C 180,E1 12243.42,E2 12243.42} C_VEL
LIN {X 0,Y 506.683,Z 780.81,A -85,B 0,C 180,E1 12248.577,E2 12248.577} C_VEL
LIN {X 0,Y 506.488,Z 780.81,A -85,B 0,C 180,E1 12253.809,E2 12253.809} C_VEL
LIN {X 0,Y 506.236,Z 780.81,A -85,B 0,C 180,E1 12259.168,E2 12259.168} C_VEL
LIN {X 0,Y 505.996,Z 780.81,A -85,B 0,C 180,E1 12264.713,E2 12264.713} C_VEL
LIN {X 0,Y 505.864,Z 780.81,A -85,B 0,C 180,E1 12270.516,E2 12270.516} C_VEL
LIN {X 0,Y 505.746,Z 780.81,A -85,B 0,C 180,E1 12276.692,E2 12276.692} C_VEL
LIN {X 0,Y 505.724,Z 780.81,A -85,B 0,C 180,E1 12278.967,E2 12278.967} C_VEL
LIN {X 0,Y 507.918,Z 786.241,A -85,B 0,C 180,E1 12279.38,E2 12279.38} C_VEL
LIN {X 0,Y 528.955,Z 820.576,A -85,B 0,C 180,E1 12282.72,E2 12282.72} C_VEL
LIN {X 0,Y 545.487,Z 856.006,A -85,B 0,C 180,E1 12285.701,E2 12285.701} C_VEL
LIN {X 0,Y 549.391,Z 867.104,A -85,B 0,C 180,E1 12286.559,E2 12286.559} C_VEL
LIN {X 0,Y 543.753,Z 910.317,A -85,B 0,C 180,E1 12288.42,E2 12288.42} C_VEL
LIN {X 0,Y 536.791,Z 952.285,A -85,B 0,C 180,E1 12291.001,E2 12291.001} C_VEL
LIN {X 0,Y 529.528,Z 989.703,A -85,B 0,C 180,E1 12294.108,E2 12294.108} C_VEL
LIN {X 0,Y 522.77,Z 1022.473,A -85,B 0,C 180,E1 12297.674,E2 12297.674} C_VEL
LIN {X 0,Y 516.693,Z 1052.012,A -85,B 0,C 180,E1 12301.851,E2 12301.851} C_VEL
LIN {X 0,Y 512.273,Z 1076.351,A -85,B 0,C 180,E1 12306.39,E2 12306.39} C_VEL
LIN {X 0,Y 509.25,Z 1096.211,A -85,B 0,C 180,E1 12311.409,E2 12311.409} C_VEL
LIN {X 0,Y 507.79,Z 1109.548,A -85,B 0,C 180,E1 12316.228,E2 12316.228} C_VEL
LIN {X 0,Y 507.264,Z 1117.225,A -85,B 0,C 180,E1 12320.571,E2 12320.571} C_VEL
LIN {X 0,Y 506.978,Z 1121.013,A -85,B 0,C 180,E1 12324.871,E2 12324.871} C_VEL
LIN {X 0,Y 507.174,Z 1120.428,A -85,B 0,C 180,E1 12330.001,E2 12330.001} C_VEL
LIN {X 0,Y 507.445,Z 1114.504,A -85,B 0,C 180,E1 12335.126,E2 12335.126} C_VEL
LIN {X 0,Y 508.433,Z 1102.96,A -85,B 0,C 180,E1 12340.273,E2 12340.273} C_VEL
LIN {X 0,Y 510.737,Z 1085.103,A -85,B 0,C 180,E1 12345.444,E2 12345.444} C_VEL
LIN {X 0,Y 514.746,Z 1061.104,A -85,B 0,C 180,E1 12350.395,E2 12350.395} C_VEL
LIN {X 0,Y 520.055,Z 1033.25,A -85,B 0,C 180,E1 12354.69,E2 12354.69} C_VEL
LIN {X 0,Y 526.269,Z 1002.049,A -85,B 0,C 180,E1 12358.388,E2 12358.388} C_VEL
LIN {X 0,Y 533.01,Z 966.786,A -85,B 0,C 180,E1 12361.61,E2 12361.61} C_VEL
LIN {X 0,Y 540.107,Z 924.609,A -85,B 0,C 180,E1 12364.485,E2 12364.485} C_VEL
LIN {X 0,Y 546.338,Z 879.026,A -85,B 0,C 180,E1 12366.678,E2 12366.678} C_VEL
LIN {X 0,Y 547.224,Z 864.813,A -85,B 0,C 180,E1 12367.256,E2 12367.256} C_VEL
LIN {X 0,Y 530.509,Z 826.209,A -85,B 0,C 180,E1 12370.214,E2 12370.214} C_VEL
LIN {X 0,Y 510.318,Z 790.361,A -85,B 0,C 180,E1 12373.192,E2 12373.192} C_VEL
LIN {X 0,Y 505.799,Z 781.588,A -85,B 0,C 180,E1 12373.886,E2 12373.886} C_VEL
LIN {X 0,Y 505.618,Z 780.81,A -85,B 0,C 180,E1 12378.896,E2 12378.896} C_VEL
LIN {X 0,Y 505.707,Z 780.81,A -85,B 0,C 180,E1 12385.411,E2 12385.411} C_VEL
LIN {X 0,Y 505.954,Z 780.81,A -85,B 0,C 180,E1 12391.456,E2 12391.456} C_VEL
LIN {X 0,Y 506.16,Z 780.81,A -85,B 0,C 180,E1 12397.744,E2 12397.744} C_VEL
LIN {X 0,Y 506.321,Z 780.81,A -85,B 0,C 180,E1 12402.756,E2 12402.756} C_VEL
LIN {X 0,Y 506.489,Z 780.81,A -85,B 0,C 180,E1 12407.945,E2 12407.945} C_VEL
LIN {X 0,Y 506.746,Z 780.81,A -85,B 0,C 180,E1 12413.148,E2 12413.148} C_VEL
LIN {X 0,Y 506.968,Z 780.81,A -85,B 0,C 180,E1 12418.29,E2 12418.29} C_VEL
LIN {X 0,Y 506.888,Z 780.81,A -85,B 0,C 180,E1 12423.415,E2 12423.415} C_VEL
LIN {X 0,Y 506.675,Z 780.81,A -85,B 0,C 180,E1 12428.572,E2 12428.572} C_VEL
LIN {X 0,Y 506.47,Z 780.81,A -85,B 0,C 180,E1 12433.804,E2 12433.804} C_VEL
LIN {X 0,Y 506.283,Z 780.81,A -85,B 0,C 180,E1 12439.161,E2 12439.161} C_VEL
LIN {X 0,Y 506.034,Z 780.81,A -85,B 0,C 180,E1 12444.705,E2 12444.705} C_VEL
LIN {X 0,Y 505.907,Z 780.81,A -85,B 0,C 180,E1 12450.507,E2 12450.507} C_VEL
LIN {X 0,Y 505.764,Z 780.81,A -85,B 0,C 180,E1 12456.684,E2 12456.684} C_VEL
LIN {X 0,Y 505.638,Z 781.071,A -85,B 0,C 180,E1 12462.545,E2 12462.545} C_VEL
LIN {X 0,Y 508.247,Z 786.682,A -85,B 0,C 180,E1 12462.959,E2 12462.959} C_VEL
LIN {X 0,Y 533.983,Z 831.561,A -85,B 0,C 180,E1 12466.527,E2 12466.527} C_VEL
LIN {X 0,Y 549.768,Z 865.418,A -85,B 0,C 180,E1 12468.838,E2 12468.838} C_VEL
LIN {X 0,Y 545.183,Z 910.237,A -85,B 0,C 180,E1 12470.238,E2 12470.238} C_VEL
LIN {X 0,Y 538.886,Z 955.877,A -85,B 0,C 180,E1 12472.417,E2 12472.417} C_VEL
LIN {X 0,Y 532.03,Z 996.547,A -85,B 0,C 180,E1 12475.137,E2 12475.137} C_VEL
LIN {X 0,Y 525.2,Z 1033.413,A -85,B 0,C 180,E1 12478.418,E2 12478.418} C_VEL
LIN {X 0,Y 519.267,Z 1064.668,A -85,B 0,C 180,E1 12482.013,E2 12482.013} C_VEL
LIN {X 0,Y 513.989,Z 1094.047,A -85,B 0,C 180,E1 12486.385,E2 12486.385} C_VEL
LIN {X 0,Y 510.23,Z 1119.066,A -85,B 0,C 180,E1 12491.353,E2 12491.353} C_VEL
LIN {X 0,Y 509.533,Z 1124.459,A -85,B 0,C 180,E1 12492.682,E2 12492.682} C_VEL
LIN {X 0,Y 507.933,Z 1127.977,A -85,B 0,C 180,E1 12493.567,E2 12493.567} C_VEL
LIN {X 0,Y 500.49,Z 1136.504,A -85,B 0,C 180,E1 12496.01,E2 12496.01} C_VEL
LIN {X 0,Y 500.325,Z 1137.236,A -85,B 0,C 180,E1 12496.247,E2 12496.247} C_VEL
LIN {X 0,Y 499.457,Z 1149.255,A -85,B 0,C 180,E1 12501.298,E2 12501.298} C_VEL
LIN {X 0,Y 499.285,Z 1154.371,A -85,B 0,C 180,E1 12504.79,E2 12504.79} C_VEL
LIN {X 0,Y 499.243,Z 1157.286,A -85,B 0,C 180,E1 12509.999,E2 12509.999} C_VEL
LIN {X 0,Y 499.28,Z 1154.374,A -85,B 0,C 180,E1 12515.208,E2 12515.208} C_VEL
LIN {X 0,Y 499.54,Z 1147.675,A -85,B 0,C 180,E1 12519.576,E2 12519.576} C_VEL
LIN {X 0,Y 500.593,Z 1134.858,A -85,B 0,C 180,E1 12524.558,E2 12524.558} C_VEL
LIN {X 0,Y 502.804,Z 1117.407,A -85,B 0,C 180,E1 12529.303,E2 12529.303} C_VEL
LIN {X 0,Y 506.871,Z 1093.067,A -85,B 0,C 180,E1 12534.199,E2 12534.199} C_VEL
LIN {X 0,Y 512.956,Z 1062.24,A -85,B 0,C 180,E1 12538.84,E2 12538.84} C_VEL
LIN {X 0,Y 520.085,Z 1027.021,A -85,B 0,C 180,E1 12542.86,E2 12542.86} C_VEL
LIN {X 0,Y 527.575,Z 989.648,A -85,B 0,C 180,E1 12546.082,E2 12546.082} C_VEL
LIN {X 0,Y 534.56,Z 951.501,A -85,B 0,C 180,E1 12548.562,E2 12548.562} C_VEL
LIN {X 0,Y 541.109,Z 908.529,A -85,B 0,C 180,E1 12550.591,E2 12550.591} C_VEL
LIN {X 0,Y 545.093,Z 867.739,A -85,B 0,C 180,E1 12551.938,E2 12551.938} C_VEL
LIN {X 0,Y 527.854,Z 831.344,A -85,B 0,C 180,E1 12554.753,E2 12554.753} C_VEL
LIN {X 0,Y 504.668,Z 792.959,A -85,B 0,C 180,E1 12558.365,E2 12558.365} C_VEL
LIN {X 0,Y 497.982,Z 782.474,A -85,B 0,C 180,E1 12559.504,E2 12559.504} C_VEL
LIN {X 0,Y 497.779,Z 780.81,A -85,B 0,C 180,E1 12559.67,E2 12559.67} C_VEL
LIN {X 0,Y 497.828,Z 780.81,A -85,B 0,C 180,E1 12565.039,E2 12565.039} C_VEL
LIN {X 0,Y 498.018,Z 780.81,A -85,B 0,C 180,E1 12571.632,E2 12571.632} C_VEL
LIN {X 0,Y 498.141,Z 780.81,A -85,B 0,C 180,E1 12576.781,E2 12576.781} C_VEL
LIN {X 0,Y 498.362,Z 780.81,A -85,B 0,C 180,E1 12582.355,E2 12582.355} C_VEL
LIN {X 0,Y 498.54,Z 780.81,A -85,B 0,C 180,E1 12587.755,E2 12587.755} C_VEL
LIN {X 0,Y 498.802,Z 780.81,A -85,B 0,C 180,E1 12593.044,E2 12593.044} C_VEL
LIN {X 0,Y 499.03,Z 780.81,A -85,B 0,C 180,E1 12598.268,E2 12598.268} C_VEL
LIN {X 0,Y 498.982,Z 780.81,A -85,B 0,C 180,E1 12603.474,E2 12603.474} C_VEL
LIN {X 0,Y 498.765,Z 780.81,A -85,B 0,C 180,E1 12608.714,E2 12608.714} C_VEL
LIN {X 0,Y 498.571,Z 780.81,A -85,B 0,C 180,E1 12614.103,E2 12614.103} C_VEL
LIN {X 0,Y 498.255,Z 780.81,A -85,B 0,C 180,E1 12619.924,E2 12619.924} C_VEL
LIN {X 0,Y 498.078,Z 780.81,A -85,B 0,C 180,E1 12625.133,E2 12625.133} C_VEL
LIN {X 0,Y 497.886,Z 780.81,A -85,B 0,C 180,E1 12631.059,E2 12631.059} C_VEL
LIN {X 0,Y 497.759,Z 780.81,A -85,B 0,C 180,E1 12637.381,E2 12637.381} C_VEL
LIN {X 0,Y 497.762,Z 780.81,A -85,B 0,C 180,E1 12637.881,E2 12637.881} C_VEL
LIN {X 0,Y 500.039,Z 786.339,A -85,B 0,C 180,E1 12638.328,E2 12638.328} C_VEL
LIN {X 0,Y 521.437,Z 820.665,A -85,B 0,C 180,E1 12641.864,E2 12641.864} C_VEL
LIN {X 0,Y 538.065,Z 855.665,A -85,B 0,C 180,E1 12644.944,E2 12644.944} C_VEL
LIN {X 0,Y 543.059,Z 871.063,A -85,B 0,C 180,E1 12646.141,E2 12646.141} C_VEL
LIN {X 0,Y 537.142,Z 913.558,A -85,B 0,C 180,E1 12648.039,E2 12648.039} C_VEL
LIN {X 0,Y 530.068,Z 954.489,A -85,B 0,C 180,E1 12650.615,E2 12650.615} C_VEL
LIN {X 0,Y 522.076,Z 993.852,A -85,B 0,C 180,E1 12653.982,E2 12653.982} C_VEL
LIN {X 0,Y 514.704,Z 1027.78,A -85,B 0,C 180,E1 12657.857,E2 12657.857} C_VEL
LIN {X 0,Y 508.544,Z 1056.386,A -85,B 0,C 180,E1 12662.145,E2 12662.145} C_VEL
LIN {X 0,Y 504.106,Z 1079.694,A -85,B 0,C 180,E1 12666.742,E2 12666.742} C_VEL
LIN {X 0,Y 501.421,Z 1097.453,A -85,B 0,C 180,E1 12671.433,E2 12671.433} C_VEL
LIN {X 0,Y 499.96,Z 1109.751,A -85,B 0,C 180,E1 12676.008,E2 12676.008} C_VEL
LIN {X 0,Y 499.377,Z 1117.454,A -85,B 0,C 180,E1 12680.421,E2 12680.421} C_VEL
LIN {X 0,Y 499.101,Z 1121.27,A -85,B 0,C 180,E1 12684.79,E2 12684.79} C_VEL
LIN {X 0,Y 499.277,Z 1120.732,A -85,B 0,C 180,E1 12690.001,E2 12690.001} C_VEL
LIN {X 0,Y 499.578,Z 1114.854,A -85,B 0,C 180,E1 12695.207,E2 12695.207} C_VEL
LIN {X 0,Y 500.626,Z 1103.355,A -85,B 0,C 180,E1 12700.435,E2 12700.435} C_VEL
LIN {X 0,Y 503.052,Z 1085.526,A -85,B 0,C 180,E1 12705.686,E2 12705.686} C_VEL
LIN {X 0,Y 507.267,Z 1061.573,A -85,B 0,C 180,E1 12710.71,E2 12710.71} C_VEL
LIN {X 0,Y 512.815,Z 1033.772,A -85,B 0,C 180,E1 12715.062,E2 12715.062} C_VEL
LIN {X 0,Y 519.317,Z 1002.603,A -85,B 0,C 180,E1 12718.807,E2 12718.807} C_VEL
LIN {X 0,Y 526.549,Z 965.997,A -85,B 0,C 180,E1 12722.174,E2 12722.174} C_VEL
LIN {X 0,Y 533.68,Z 925.033,A -85,B 0,C 180,E1 12724.986,E2 12724.986} C_VEL
LIN {X 0,Y 540.093,Z 879.978,A -85,B 0,C 180,E1 12727.173,E2 12727.173} C_VEL
LIN {X 0,Y 540.839,Z 867.736,A -85,B 0,C 180,E1 12727.685,E2 12727.685} C_VEL
LIN {X 0,Y 524.548,Z 829.445,A -85,B 0,C 180,E1 12730.719,E2 12730.719} C_VEL
LIN {X 0,Y 503.757,Z 792.15,A -85,B 0,C 180,E1 12733.913,E2 12733.913} C_VEL
LIN {X 0,Y 497.927,Z 782.362,A -85,B 0,C 180,E1 12734.812,E2 12734.812} C_VEL
LIN {X 0,Y 497.743,Z 780.81,A -85,B 0,C 180,E1 12734.946,E2 12734.946} C_VEL
LIN {X 0,Y 497.685,Z 780.81,A -85,B 0,C 180,E1 12740.39,E2 12740.39} C_VEL
LIN {X 0,Y 497.822,Z 780.81,A -85,B 0,C 180,E1 12746.884,E2 12746.884} C_VEL
LIN {X 0,Y 498.054,Z 780.81,A -85,B 0,C 180,E1 12752.931,E2 12752.931} C_VEL
LIN {X 0,Y 498.249,Z 780.81,A -85,B 0,C 180,E1 12758.659,E2 12758.659} C_VEL
LIN {X 0,Y 498.421,Z 780.81,A -85,B 0,C 180,E1 12764.165,E2 12764.165} C_VEL
LIN {X 0,Y 498.666,Z 780.81,A -85,B 0,C 180,E1 12769.523,E2 12769.523} C_VEL
LIN {X 0,Y 498.914,Z 780.81,A -85,B 0,C 180,E1 12774.785,E2 12774.785} C_VEL
LIN {X 0,Y 499.244,Z 780.81,A -85,B 0,C 180,E1 12779.997,E2 12779.997} C_VEL
LIN {X 0,Y 498.932,Z 780.81,A -85,B 0,C 180,E1 12785.21,E2 12785.21} C_VEL
LIN {X 0,Y 498.687,Z 780.81,A -85,B 0,C 180,E1 12790.471,E2 12790.471} C_VEL
LIN {X 0,Y 498.468,Z 780.81,A -85,B 0,C 180,E1 12795.827,E2 12795.827} C_VEL
LIN {X 0,Y 498.259,Z 780.81,A -85,B 0,C 180,E1 12801.335,E2 12801.335} C_VEL
LIN {X 0,Y 498.061,Z 780.81,A -85,B 0,C 180,E1 12807.063,E2 12807.063} C_VEL
LIN {X 0,Y 497.921,Z 780.81,A -85,B 0,C 180,E1 12813.102,E2 12813.102} C_VEL
LIN {X 0,Y 497.671,Z 780.81,A -85,B 0,C 180,E1 12819.604,E2 12819.604} C_VEL
LIN {X 0,Y 497.7,Z 781.373,A -85,B 0,C 180,E1 12821.599,E2 12821.599} C_VEL
LIN {X 0,Y 500.405,Z 786.752,A -85,B 0,C 180,E1 12822.038,E2 12822.038} C_VEL
LIN {X 0,Y 525.347,Z 829.587,A -85,B 0,C 180,E1 12825.631,E2 12825.631} C_VEL
LIN {X 0,Y 543.308,Z 867.844,A -85,B 0,C 180,E1 12828.354,E2 12828.354} C_VEL
LIN {X 0,Y 538.61,Z 912.5,A -85,B 0,C 180,E1 12829.812,E2 12829.812} C_VEL
LIN {X 0,Y 532.484,Z 955.306,A -85,B 0,C 180,E1 12831.885,E2 12831.885} C_VEL
LIN {X 0,Y 525.34,Z 996.032,A -85,B 0,C 180,E1 12834.627,E2 12834.627} C_VEL
LIN {X 0,Y 518.233,Z 1032.937,A -85,B 0,C 180,E1 12837.941,E2 12837.941} C_VEL
LIN {X 0,Y 512.043,Z 1064.26,A -85,B 0,C 180,E1 12841.583,E2 12841.583} C_VEL
LIN {X 0,Y 506.5,Z 1093.676,A -85,B 0,C 180,E1 12846.014,E2 12846.014} C_VEL
LIN {X 0,Y 502.525,Z 1118.722,A -85,B 0,C 180,E1 12851.057,E2 12851.057} C_VEL
LIN {X 0,Y 500.325,Z 1137.236,A -85,B 0,C 180,E1 12856.247,E2 12856.247} C_VEL
LIN {X 0,Y 495.919,Z 1142.421,A -85,B 0,C 180,E1 12858.104,E2 12858.104} C_VEL
LIN {X 0,Y 491.688,Z 1146.803,A -85,B 0,C 180,E1 12860.021,E2 12860.021} C_VEL
LIN {X 0,Y 491.386,Z 1154.08,A -85,B 0,C 180,E1 12864.706,E2 12864.706} C_VEL
LIN {X 0,Y 491.39,Z 1156.663,A -85,B 0,C 180,E1 12868.237,E2 12868.237} C_VEL
LIN {X 0,Y 491.371,Z 1156.662,A -85,B 0,C 180,E1 12871.761,E2 12871.761} C_VEL
LIN {X 0,Y 491.464,Z 1151.877,A -85,B 0,C 180,E1 12877.064,E2 12877.064} C_VEL
LIN {X 0,Y 492.038,Z 1142.456,A -85,B 0,C 180,E1 12881.963,E2 12881.963} C_VEL
LIN {X 0,Y 493.831,Z 1126.089,A -85,B 0,C 180,E1 12887.357,E2 12887.357} C_VEL
LIN {X 0,Y 497.236,Z 1104.107,A -85,B 0,C 180,E1 12892.46,E2 12892.46} C_VEL
LIN {X 0,Y 502.349,Z 1077.673,A -85,B 0,C 180,E1 12897.063,E2 12897.063} C_VEL
LIN {X 0,Y 508.807,Z 1047.86,A -85,B 0,C 180,E1 12901.064,E2 12901.064} C_VEL
LIN {X 0,Y 516.508,Z 1011.968,A -85,B 0,C 180,E1 12904.771,E2 12904.771} C_VEL
LIN {X 0,Y 524.919,Z 970.272,A -85,B 0,C 180,E1 12907.97,E2 12907.97} C_VEL
LIN {X 0,Y 532.503,Z 925.791,A -85,B 0,C 180,E1 12910.424,E2 12910.424} C_VEL
LIN {X 0,Y 538.423,Z 880.855,A -85,B 0,C 180,E1 12912.101,E2 12912.101} C_VEL
LIN {X 0,Y 538.955,Z 870.405,A -85,B 0,C 180,E1 12912.448,E2 12912.448} C_VEL
LIN {X 0,Y 521.971,Z 834.302,A -85,B 0,C 180,E1 12915.35,E2 12915.35} C_VEL
LIN {X 0,Y 500.322,Z 798.459,A -85,B 0,C 180,E1 12918.829,E2 12918.829} C_VEL
LIN {X 0,Y 490.016,Z 782.494,A -85,B 0,C 180,E1 12920.65,E2 12920.65} C_VEL
LIN {X 0,Y 489.831,Z 780.81,A -85,B 0,C 180,E1 12920.743,E2 12920.743} C_VEL
LIN {X 0,Y 489.914,Z 780.81,A -85,B 0,C 180,E1 12926.385,E2 12926.385} C_VEL
LIN {X 0,Y 490.134,Z 780.81,A -85,B 0,C 180,E1 12932.462,E2 12932.462} C_VEL
LIN {X 0,Y 490.278,Z 780.81,A -85,B 0,C 180,E1 12938.3,E2 12938.3} C_VEL
LIN {X 0,Y 490.474,Z 780.81,A -85,B 0,C 180,E1 12943.908,E2 12943.908} C_VEL
LIN {X 0,Y 490.724,Z 780.81,A -85,B 0,C 180,E1 12950.187,E2 12950.187} C_VEL
LIN {X 0,Y 491.151,Z 780.81,A -85,B 0,C 180,E1 12956.475,E2 12956.475} C_VEL
LIN {X 0,Y 491.25,Z 780.81,A -85,B 0,C 180,E1 12961.765,E2 12961.765} C_VEL
LIN {X 0,Y 490.944,Z 780.81,A -85,B 0,C 180,E1 12967.074,E2 12967.074} C_VEL
LIN {X 0,Y 490.658,Z 780.81,A -85,B 0,C 180,E1 12972.45,E2 12972.45} C_VEL
LIN {X 0,Y 490.436,Z 780.81,A -85,B 0,C 180,E1 12977.945,E2 12977.945} C_VEL
LIN {X 0,Y 490.184,Z 780.81,A -85,B 0,C 180,E1 12983.624,E2 12983.624} C_VEL
LIN {X 0,Y 490.015,Z 780.81,A -85,B 0,C 180,E1 12989.562,E2 12989.562} C_VEL
LIN {X 0,Y 489.841,Z 780.81,A -85,B 0,C 180,E1 12995.879,E2 12995.879} C_VEL
LIN {X 0,Y 489.809,Z 780.81,A -85,B 0,C 180,E1 12996.729,E2 12996.729} C_VEL
LIN {X 0,Y 492.036,Z 786.277,A -85,B 0,C 180,E1 12997.195,E2 12997.195} C_VEL
LIN {X 0,Y 511.505,Z 816.398,A -85,B 0,C 180,E1 13000.531,E2 13000.531} C_VEL
LIN {X 0,Y 529.202,Z 851.855,A -85,B 0,C 180,E1 13003.849,E2 13003.849} C_VEL
LIN {X 0,Y 536.946,Z 873.472,A -85,B 0,C 180,E1 13005.656,E2 13005.656} C_VEL
LIN {X 0,Y 530.897,Z 914.895,A -85,B 0,C 180,E1 13007.545,E2 13007.545} C_VEL
LIN {X 0,Y 523.52,Z 955.725,A -85,B 0,C 180,E1 13010.153,E2 13010.153} C_VEL
LIN {X 0,Y 515.284,Z 994.677,A -85,B 0,C 180,E1 13013.531,E2 13013.531} C_VEL
LIN {X 0,Y 507.391,Z 1029.526,A -85,B 0,C 180,E1 13017.584,E2 13017.584} C_VEL
LIN {X 0,Y 500.791,Z 1058.848,A -85,B 0,C 180,E1 13022.116,E2 13022.116} C_VEL
LIN {X 0,Y 496.334,Z 1081.171,A -85,B 0,C 180,E1 13026.686,E2 13026.686} C_VEL
LIN {X 0,Y 493.509,Z 1099.19,A -85,B 0,C 180,E1 13031.639,E2 13031.639} C_VEL
LIN {X 0,Y 492.003,Z 1111.846,A -85,B 0,C 180,E1 13036.683,E2 13036.683} C_VEL
LIN {X 0,Y 491.406,Z 1118.824,A -85,B 0,C 180,E1 13041.157,E2 13041.157} C_VEL
LIN {X 0,Y 491.254,Z 1121.956,A -85,B 0,C 180,E1 13046.474,E2 13046.474} C_VEL
LIN {X 0,Y 491.495,Z 1119.688,A -85,B 0,C 180,E1 13051.763,E2 13051.763} C_VEL
LIN {X 0,Y 491.804,Z 1113.682,A -85,B 0,C 180,E1 13056.175,E2 13056.175} C_VEL
LIN {X 0,Y 493.083,Z 1101.649,A -85,B 0,C 180,E1 13061.318,E2 13061.318} C_VEL
LIN {X 0,Y 495.66,Z 1084.058,A -85,B 0,C 180,E1 13066.4,E2 13066.4} C_VEL
LIN {X 0,Y 500.074,Z 1060.827,A -85,B 0,C 180,E1 13071.262,E2 13071.262} C_VEL
LIN {X 0,Y 506.303,Z 1031.171,A -85,B 0,C 180,E1 13075.882,E2 13075.882} C_VEL
LIN {X 0,Y 513.57,Z 997.431,A -85,B 0,C 180,E1 13079.839,E2 13079.839} C_VEL
LIN {X 0,Y 520.699,Z 962.339,A -85,B 0,C 180,E1 13082.973,E2 13082.973} C_VEL
LIN {X 0,Y 527.552,Z 923.969,A -85,B 0,C 180,E1 13085.58,E2 13085.58} C_VEL
LIN {X 0,Y 534.069,Z 879.32,A -85,B 0,C 180,E1 13087.749,E2 13087.749} C_VEL
LIN {X 0,Y 534.422,Z 870.594,A -85,B 0,C 180,E1 13088.133,E2 13088.133} C_VEL
LIN {X 0,Y 518.355,Z 832.06,A -85,B 0,C 180,E1 13091.28,E2 13091.28} C_VEL
LIN {X 0,Y 496.741,Z 793.143,A -85,B 0,C 180,E1 13094.735,E2 13094.735} C_VEL
LIN {X 0,Y 489.902,Z 781.902,A -85,B 0,C 180,E1 13095.831,E2 13095.831} C_VEL
LIN {X 0,Y 489.832,Z 780.81,A -85,B 0,C 180,E1 13095.904,E2 13095.904} C_VEL
LIN {X 0,Y 489.761,Z 780.81,A -85,B 0,C 180,E1 13101.901,E2 13101.901} C_VEL
LIN {X 0,Y 489.943,Z 780.81,A -85,B 0,C 180,E1 13108.38,E2 13108.38} C_VEL
LIN {X 0,Y 490.142,Z 780.81,A -85,B 0,C 180,E1 13114.431,E2 13114.431} C_VEL
LIN {X 0,Y 490.406,Z 780.81,A -85,B 0,C 180,E1 13120.188,E2 13120.188} C_VEL
LIN {X 0,Y 490.581,Z 780.81,A -85,B 0,C 180,E1 13125.734,E2 13125.734} C_VEL
LIN {X 0,Y 490.847,Z 780.81,A -85,B 0,C 180,E1 13131.144,E2 13131.144} C_VEL
LIN {X 0,Y 491.173,Z 780.81,A -85,B 0,C 180,E1 13136.47,E2 13136.47} C_VEL
LIN {X 0,Y 491.266,Z 780.81,A -85,B 0,C 180,E1 13141.76,E2 13141.76} C_VEL
LIN {X 0,Y 490.901,Z 780.81,A -85,B 0,C 180,E1 13147.069,E2 13147.069} C_VEL
LIN {X 0,Y 490.652,Z 780.81,A -85,B 0,C 180,E1 13152.445,E2 13152.445} C_VEL
LIN {X 0,Y 490.479,Z 780.81,A -85,B 0,C 180,E1 13157.938,E2 13157.938} C_VEL
LIN {X 0,Y 490.219,Z 780.81,A -85,B 0,C 180,E1 13163.616,E2 13163.616} C_VEL
LIN {X 0,Y 490.052,Z 780.81,A -85,B 0,C 180,E1 13169.554,E2 13169.554} C_VEL
LIN {X 0,Y 489.874,Z 780.81,A -85,B 0,C 180,E1 13175.869,E2 13175.869} C_VEL
LIN {X 0,Y 489.753,Z 780.81,A -85,B 0,C 180,E1 13180.567,E2 13180.567} C_VEL
LIN {X 0,Y 492.239,Z 786.534,A -85,B 0,C 180,E1 13181.025,E2 13181.025} C_VEL
LIN {X 0,Y 515.234,Z 824.91,A -85,B 0,C 180,E1 13184.475,E2 13184.475} C_VEL
LIN {X 0,Y 534.15,Z 863.787,A -85,B 0,C 180,E1 13187.386,E2 13187.386} C_VEL
LIN {X 0,Y 536.985,Z 872.666,A -85,B 0,C 180,E1 13187.947,E2 13187.947} C_VEL
LIN {X 0,Y 531.736,Z 917.119,A -85,B 0,C 180,E1 13189.474,E2 13189.474} C_VEL
LIN {X 0,Y 525.515,Z 958.187,A -85,B 0,C 180,E1 13191.55,E2 13191.55} C_VEL
LIN {X 0,Y 518.229,Z 998.326,A -85,B 0,C 180,E1 13194.324,E2 13194.324} C_VEL
LIN {X 0,Y 510.416,Z 1037.013,A -85,B 0,C 180,E1 13197.923,E2 13197.923} C_VEL
LIN {X 0,Y 503.381,Z 1071.178,A -85,B 0,C 180,E1 13202.148,E2 13202.148} C_VEL
LIN {X 0,Y 497.832,Z 1099.427,A -85,B 0,C 180,E1 13206.758,E2 13206.758} C_VEL
LIN {X 0,Y 494.488,Z 1120.496,A -85,B 0,C 180,E1 13211.284,E2 13211.284} C_VEL
LIN {X 0,Y 492.428,Z 1137.574,A -85,B 0,C 180,E1 13216.241,E2 13216.241} C_VEL
LIN {X 0,Y 491.688,Z 1146.803,A -85,B 0,C 180,E1 13220.021,E2 13220.021} C_VEL
LIN {X 0,Y 489.07,Z 1149.644,A -85,B 0,C 180,E1 13221.486,E2 13221.486} C_VEL
LIN {X 0,Y 483.631,Z 1152.768,A -85,B 0,C 180,E1 13223.71,E2 13223.71} C_VEL
LIN {X 0,Y 483.517,Z 1153.058,A -85,B 0,C 180,E1 13223.969,E2 13223.969} C_VEL
LIN {X 0,Y 483.515,Z 1156.38,A -85,B 0,C 180,E1 13228.208,E2 13228.208} C_VEL
LIN {X 0,Y 483.475,Z 1156.383,A -85,B 0,C 180,E1 13231.79,E2 13231.79} C_VEL
LIN {X 0,Y 483.568,Z 1151.61,A -85,B 0,C 180,E1 13237.179,E2 13237.179} C_VEL
LIN {X 0,Y 484.179,Z 1142.204,A -85,B 0,C 180,E1 13242.16,E2 13242.16} C_VEL
LIN {X 0,Y 486.066,Z 1125.85,A -85,B 0,C 180,E1 13247.644,E2 13247.644} C_VEL
LIN {X 0,Y 489.624,Z 1104.161,A -85,B 0,C 180,E1 13252.77,E2 13252.77} C_VEL
LIN {X 0,Y 494.777,Z 1078.97,A -85,B 0,C 180,E1 13257.264,E2 13257.264} C_VEL
LIN {X 0,Y 501.828,Z 1047.725,A -85,B 0,C 180,E1 13261.546,E2 13261.546} C_VEL
LIN {X 0,Y 510.147,Z 1010.885,A -85,B 0,C 180,E1 13265.374,E2 13265.374} C_VEL
LIN {X 0,Y 518.643,Z 970.193,A -85,B 0,C 180,E1 13268.518,E2 13268.518} C_VEL
LIN {X 0,Y 526.255,Z 927.091,A -85,B 0,C 180,E1 13270.928,E2 13270.928} C_VEL
LIN {X 0,Y 532.363,Z 883.133,A -85,B 0,C 180,E1 13272.608,E2 13272.608} C_VEL
LIN {X 0,Y 532.93,Z 873.26,A -85,B 0,C 180,E1 13272.957,E2 13272.957} C_VEL
LIN {X 0,Y 515.617,Z 836.174,A -85,B 0,C 180,E1 13276.049,E2 13276.049} C_VEL
LIN {X 0,Y 493.14,Z 799.185,A -85,B 0,C 180,E1 13279.814,E2 13279.814} C_VEL
LIN {X 0,Y 484.144,Z 786.299,A -85,B 0,C 180,E1 13281.449,E2 13281.449} C_VEL
LIN {X 0,Y 481.893,Z 780.81,A -85,B 0,C 180,E1 13282.04,E2 13282.04} C_VEL
LIN {X 0,Y 482.002,Z 780.81,A -85,B 0,C 180,E1 13287.827,E2 13287.827} C_VEL
LIN {X 0,Y 482.22,Z 780.81,A -85,B 0,C 180,E1 13293.986,E2 13293.986} C_VEL
LIN {X 0,Y 482.459,Z 780.81,A -85,B 0,C 180,E1 13299.986,E2 13299.986} C_VEL
LIN {X 0,Y 482.703,Z 780.81,A -85,B 0,C 180,E1 13306.034,E2 13306.034} C_VEL
LIN {X 0,Y 482.917,Z 780.81,A -85,B 0,C 180,E1 13311.003,E2 13311.003} C_VEL
LIN {X 0,Y 483.256,Z 780.81,A -85,B 0,C 180,E1 13316.418,E2 13316.418} C_VEL
LIN {X 0,Y 483.349,Z 780.81,A -85,B 0,C 180,E1 13321.794,E2 13321.794} C_VEL
LIN {X 0,Y 483.025,Z 780.81,A -85,B 0,C 180,E1 13327.19,E2 13327.19} C_VEL
LIN {X 0,Y 482.761,Z 780.81,A -85,B 0,C 180,E1 13333.994,E2 13333.994} C_VEL
LIN {X 0,Y 482.46,Z 780.81,A -85,B 0,C 180,E1 13340.152,E2 13340.152} C_VEL
LIN {X 0,Y 482.209,Z 780.81,A -85,B 0,C 180,E1 13346.02,E2 13346.02} C_VEL
LIN {X 0,Y 482.024,Z 780.81,A -85,B 0,C 180,E1 13352.201,E2 13352.201} C_VEL
LIN {X 0,Y 481.944,Z 781.328,A -85,B 0,C 180,E1 13355.55,E2 13355.55} C_VEL
LIN {X 0,Y 484.609,Z 786.744,A -85,B 0,C 180,E1 13356.095,E2 13356.095} C_VEL
LIN {X 0,Y 504.709,Z 817.959,A -85,B 0,C 180,E1 13359.715,E2 13359.715} C_VEL
LIN {X 0,Y 521.995,Z 852.147,A -85,B 0,C 180,E1 13363.067,E2 13363.067} C_VEL
LIN {X 0,Y 530.726,Z 874.967,A -85,B 0,C 180,E1 13365.098,E2 13365.098} C_VEL
LIN {X 0,Y 524.608,Z 916.589,A -85,B 0,C 180,E1 13367.056,E2 13367.056} C_VEL
LIN {X 0,Y 517.197,Z 956.199,A -85,B 0,C 180,E1 13369.623,E2 13369.623} C_VEL
LIN {X 0,Y 508.674,Z 994.985,A -85,B 0,C 180,E1 13373.019,E2 13373.019} C_VEL
LIN {X 0,Y 500.495,Z 1029.561,A -85,B 0,C 180,E1 13377.082,E2 13377.082} C_VEL
LIN {X 0,Y 493.548,Z 1058.941,A -85,B 0,C 180,E1 13381.67,E2 13381.67} C_VEL
LIN {X 0,Y 488.815,Z 1081.312,A -85,B 0,C 180,E1 13386.306,E2 13386.306} C_VEL
LIN {X 0,Y 485.775,Z 1099.375,A -85,B 0,C 180,E1 13391.336,E2 13391.336} C_VEL
LIN {X 0,Y 484.147,Z 1112.056,A -85,B 0,C 180,E1 13396.463,E2 13396.463} C_VEL
LIN {X 0,Y 483.531,Z 1119.073,A -85,B 0,C 180,E1 13401.011,E2 13401.011} C_VEL
LIN {X 0,Y 483.35,Z 1122.231,A -85,B 0,C 180,E1 13406.416,E2 13406.416} C_VEL
LIN {X 0,Y 483.606,Z 1120.003,A -85,B 0,C 180,E1 13411.792,E2 13411.792} C_VEL
LIN {X 0,Y 483.945,Z 1114.026,A -85,B 0,C 180,E1 13416.275,E2 13416.275} C_VEL
LIN {X 0,Y 485.303,Z 1102.035,A -85,B 0,C 180,E1 13421.502,E2 13421.502} C_VEL
LIN {X 0,Y 487.986,Z 1084.57,A -85,B 0,C 180,E1 13426.646,E2 13426.646} C_VEL
LIN {X 0,Y 492.886,Z 1060.049,A -85,B 0,C 180,E1 13431.824,E2 13431.824} C_VEL
LIN {X 0,Y 499.539,Z 1030.1,A -85,B 0,C 180,E1 13436.5,E2 13436.5} C_VEL
LIN {X 0,Y 507.529,Z 994.451,A -85,B 0,C 180,E1 13440.657,E2 13440.657} C_VEL
LIN {X 0,Y 515.734,Z 955.035,A -85,B 0,C 180,E1 13444.07,E2 13444.07} C_VEL
LIN {X 0,Y 523.016,Z 913.58,A -85,B 0,C 180,E1 13446.707,E2 13446.707} C_VEL
LIN {X 0,Y 528.235,Z 873.872,A -85,B 0,C 180,E1 13448.553,E2 13448.553} C_VEL
LIN {X 0,Y 512.393,Z 835.267,A -85,B 0,C 180,E1 13451.799,E2 13451.799} C_VEL
LIN {X 0,Y 491.944,Z 798.273,A -85,B 0,C 180,E1 13455.224,E2 13455.224} C_VEL
LIN {X 0,Y 482.089,Z 782.62,A -85,B 0,C 180,E1 13456.85,E2 13456.85} C_VEL
LIN {X 0,Y 481.882,Z 780.81,A -85,B 0,C 180,E1 13456.974,E2 13456.974} C_VEL
LIN {X 0,Y 481.867,Z 780.81,A -85,B 0,C 180,E1 13463.432,E2 13463.432} C_VEL
LIN {X 0,Y 482.089,Z 780.81,A -85,B 0,C 180,E1 13469.902,E2 13469.902} C_VEL
LIN {X 0,Y 482.246,Z 780.81,A -85,B 0,C 180,E1 13475.963,E2 13475.963} C_VEL
LIN {X 0,Y 482.482,Z 780.81,A -85,B 0,C 180,E1 13481.749,E2 13481.749} C_VEL
LIN {X 0,Y 482.702,Z 780.81,A -85,B 0,C 180,E1 13487.341,E2 13487.341} C_VEL
LIN {X 0,Y 482.982,Z 780.81,A -85,B 0,C 180,E1 13493.133,E2 13493.133} C_VEL
LIN {X 0,Y 483.305,Z 780.81,A -85,B 0,C 180,E1 13498.206,E2 13498.206} C_VEL
LIN {X 0,Y 483.183,Z 780.81,A -85,B 0,C 180,E1 13503.583,E2 13503.583} C_VEL
LIN {X 0,Y 482.938,Z 780.81,A -85,B 0,C 180,E1 13508.997,E2 13508.997} C_VEL
LIN {X 0,Y 482.684,Z 780.81,A -85,B 0,C 180,E1 13514.499,E2 13514.499} C_VEL
LIN {X 0,Y 482.477,Z 780.81,A -85,B 0,C 180,E1 13520.146,E2 13520.146} C_VEL
LIN {X 0,Y 482.236,Z 780.81,A -85,B 0,C 180,E1 13526.013,E2 13526.013} C_VEL
LIN {X 0,Y 482.066,Z 780.81,A -85,B 0,C 180,E1 13532.191,E2 13532.191} C_VEL
LIN {X 0,Y 481.858,Z 780.81,A -85,B 0,C 180,E1 13538.832,E2 13538.832} C_VEL
LIN {X 0,Y 481.912,Z 781.441,A -85,B 0,C 180,E1 13539.559,E2 13539.559} C_VEL
LIN {X 0,Y 484.561,Z 786.776,A -85,B 0,C 180,E1 13540.033,E2 13540.033} C_VEL
LIN {X 0,Y 508.346,Z 826.161,A -85,B 0,C 180,E1 13543.749,E2 13543.749} C_VEL
LIN {X 0,Y 526.794,Z 863.891,A -85,B 0,C 180,E1 13546.693,E2 13546.693} C_VEL
LIN {X 0,Y 530.78,Z 874.638,A -85,B 0,C 180,E1 13547.443,E2 13547.443} C_VEL
LIN {X 0,Y 525.074,Z 920.25,A -85,B 0,C 180,E1 13549.063,E2 13549.063} C_VEL
LIN {X 0,Y 518.583,Z 961.06,A -85,B 0,C 180,E1 13551.207,E2 13551.207} C_VEL
LIN {X 0,Y 511.356,Z 999.034,A -85,B 0,C 180,E1 13553.892,E2 13553.892} C_VEL
LIN {X 0,Y 503.283,Z 1037.606,A -85,B 0,C 180,E1 13557.54,E2 13557.54} C_VEL
LIN {X 0,Y 495.753,Z 1072.572,A -85,B 0,C 180,E1 13561.96,E2 13561.96} C_VEL
LIN {X 0,Y 489.951,Z 1101.328,A -85,B 0,C 180,E1 13566.809,E2 13566.809} C_VEL
LIN {X 0,Y 486.229,Z 1123.693,A -85,B 0,C 180,E1 13571.893,E2 13571.893} C_VEL
LIN {X 0,Y 484.35,Z 1139.664,A -85,B 0,C 180,E1 13576.926,E2 13576.926} C_VEL
LIN {X 0,Y 483.645,Z 1150.247,A -85,B 0,C 180,E1 13581.916,E2 13581.916} C_VEL
LIN {X 0,Y 483.517,Z 1153.058,A -85,B 0,C 180,E1 13583.969,E2 13583.969} C_VEL
LIN {X 0,Y 482.186,Z 1154.152,A -85,B 0,C 180,E1 13584.987,E2 13584.987} C_VEL
LIN {X 0,Y 475.65,Z 1155.931,A -85,B 0,C 180,E1 13587.777,E2 13587.777} C_VEL
LIN {X 0,Y 475.593,Z 1156.022,A -85,B 0,C 180,E1 13588.042,E2 13588.042} C_VEL
LIN {X 0,Y 475.574,Z 1156.104,A -85,B 0,C 180,E1 13591.82,E2 13591.82} C_VEL
LIN {X 0,Y 475.674,Z 1151.344,A -85,B 0,C 180,E1 13597.299,E2 13597.299} C_VEL
LIN {X 0,Y 476.339,Z 1141.955,A -85,B 0,C 180,E1 13602.364,E2 13602.364} C_VEL
LIN {X 0,Y 478.303,Z 1125.614,A -85,B 0,C 180,E1 13607.94,E2 13607.94} C_VEL
LIN {X 0,Y 482.025,Z 1104.314,A -85,B 0,C 180,E1 13613.069,E2 13613.069} C_VEL
LIN {X 0,Y 487.513,Z 1078.795,A -85,B 0,C 180,E1 13617.705,E2 13617.705} C_VEL
LIN {X 0,Y 494.922,Z 1047.594,A -85,B 0,C 180,E1 13622.038,E2 13622.038} C_VEL
LIN {X 0,Y 503.579,Z 1010.844,A -85,B 0,C 180,E1 13625.903,E2 13625.903} C_VEL
LIN {X 0,Y 512.414,Z 970.173,A -85,B 0,C 180,E1 13629.074,E2 13629.074} C_VEL
LIN {X 0,Y 520.126,Z 928.034,A -85,B 0,C 180,E1 13631.46,E2 13631.46} C_VEL
LIN {X 0,Y 526.417,Z 884.973,A -85,B 0,C 180,E1 13633.14,E2 13633.14} C_VEL
LIN {X 0,Y 526.953,Z 876.156,A -85,B 0,C 180,E1 13633.467,E2 13633.467} C_VEL
LIN {X 0,Y 510.374,Z 840.318,A -85,B 0,C 180,E1 13636.584,E2 13636.584} C_VEL
LIN {X 0,Y 489.424,Z 805.339,A -85,B 0,C 180,E1 13640.21,E2 13640.21} C_VEL
LIN {X 0,Y 476.445,Z 786.526,A -85,B 0,C 180,E1 13642.669,E2 13642.669} C_VEL
LIN {X 0,Y 474.066,Z 781.808,A -85,B 0,C 180,E1 13643.182,E2 13643.182} C_VEL
LIN {X 0,Y 474.007,Z 780.81,A -85,B 0,C 180,E1 13643.335,E2 13643.335} C_VEL
LIN {X 0,Y 474.126,Z 780.81,A -85,B 0,C 180,E1 13649.374,E2 13649.374} C_VEL
LIN {X 0,Y 474.31,Z 780.81,A -85,B 0,C 180,E1 13655.541,E2 13655.541} C_VEL
LIN {X 0,Y 474.552,Z 780.81,A -85,B 0,C 180,E1 13661.438,E2 13661.438} C_VEL
LIN {X 0,Y 474.791,Z 780.81,A -85,B 0,C 180,E1 13667.132,E2 13667.132} C_VEL
LIN {X 0,Y 475.052,Z 780.81,A -85,B 0,C 180,E1 13672.694,E2 13672.694} C_VEL
LIN {X 0,Y 475.364,Z 780.81,A -85,B 0,C 180,E1 13678.181,E2 13678.181} C_VEL
LIN {X 0,Y 475.27,Z 780.81,A -85,B 0,C 180,E1 13683.648,E2 13683.648} C_VEL
LIN {X 0,Y 474.967,Z 780.81,A -85,B 0,C 180,E1 13689.514,E2 13689.514} C_VEL
LIN {X 0,Y 474.774,Z 780.81,A -85,B 0,C 180,E1 13694.752,E2 13694.752} C_VEL
LIN {X 0,Y 474.493,Z 780.81,A -85,B 0,C 180,E1 13700.506,E2 13700.506} C_VEL
LIN {X 0,Y 474.206,Z 780.81,A -85,B 0,C 180,E1 13706.845,E2 13706.845} C_VEL
LIN {X 0,Y 474.03,Z 780.81,A -85,B 0,C 180,E1 13712.812,E2 13712.812} C_VEL
LIN {X 0,Y 474.087,Z 781.531,A -85,B 0,C 180,E1 13714.276,E2 13714.276} C_VEL
LIN {X 0,Y 476.749,Z 786.761,A -85,B 0,C 180,E1 13714.849,E2 13714.849} C_VEL
LIN {X 0,Y 497.046,Z 817.864,A -85,B 0,C 180,E1 13718.688,E2 13718.688} C_VEL
LIN {X 0,Y 514.134,Z 850.877,A -85,B 0,C 180,E1 13722.102,E2 13722.102} C_VEL
LIN {X 0,Y 524.722,Z 879.115,A -85,B 0,C 180,E1 13724.68,E2 13724.68} C_VEL
LIN {X 0,Y 517.535,Z 922.789,A -85,B 0,C 180,E1 13726.807,E2 13726.807} C_VEL
LIN {X 0,Y 509.813,Z 961.49,A -85,B 0,C 180,E1 13729.456,E2 13729.456} C_VEL
LIN {X 0,Y 501.622,Z 997.087,A -85,B 0,C 180,E1 13732.682,E2 13732.682} C_VEL
LIN {X 0,Y 493.206,Z 1031.284,A -85,B 0,C 180,E1 13736.792,E2 13736.792} C_VEL
LIN {X 0,Y 485.725,Z 1061.63,A -85,B 0,C 180,E1 13741.679,E2 13741.679} C_VEL
LIN {X 0,Y 480.558,Z 1085.313,A -85,B 0,C 180,E1 13746.856,E2 13746.856} C_VEL
LIN {X 0,Y 477.622,Z 1102.394,A -85,B 0,C 180,E1 13752.034,E2 13752.034} C_VEL
LIN {X 0,Y 476.106,Z 1114.004,A -85,B 0,C 180,E1 13757.164,E2 13757.164} C_VEL
LIN {X 0,Y 475.661,Z 1119.321,A -85,B 0,C 180,E1 13760.861,E2 13760.861} C_VEL
LIN {X 0,Y 475.447,Z 1122.505,A -85,B 0,C 180,E1 13766.357,E2 13766.357} C_VEL
LIN {X 0,Y 475.713,Z 1120.318,A -85,B 0,C 180,E1 13771.821,E2 13771.821} C_VEL
LIN {X 0,Y 476.104,Z 1114.367,A -85,B 0,C 180,E1 13776.379,E2 13776.379} C_VEL
LIN {X 0,Y 477.393,Z 1103.347,A -85,B 0,C 180,E1 13781.365,E2 13781.365} C_VEL
LIN {X 0,Y 480.015,Z 1086.775,A -85,B 0,C 180,E1 13786.46,E2 13786.46} C_VEL
LIN {X 0,Y 484.657,Z 1064.055,A -85,B 0,C 180,E1 13791.498,E2 13791.498} C_VEL
LIN {X 0,Y 490.472,Z 1038.507,A -85,B 0,C 180,E1 13795.787,E2 13795.787} C_VEL
LIN {X 0,Y 497.975,Z 1006.887,A -85,B 0,C 180,E1 13799.855,E2 13799.855} C_VEL
LIN {X 0,Y 506.384,Z 969.296,A -85,B 0,C 180,E1 13803.493,E2 13803.493} C_VEL
LIN {X 0,Y 514.513,Z 927.269,A -85,B 0,C 180,E1 13806.495,E2 13806.495} C_VEL
LIN {X 0,Y 521.363,Z 884.275,A -85,B 0,C 180,E1 13808.666,E2 13808.666} C_VEL
LIN {X 0,Y 521.86,Z 876.436,A -85,B 0,C 180,E1 13809.039,E2 13809.039} C_VEL
LIN {X 0,Y 506.213,Z 837.984,A -85,B 0,C 180,E1 13812.376,E2 13812.376} C_VEL
LIN {X 0,Y 486.904,Z 802.85,A -85,B 0,C 180,E1 13815.761,E2 13815.761} C_VEL
LIN {X 0,Y 474.066,Z 782.009,A -85,B 0,C 180,E1 13817.986,E2 13817.986} C_VEL
LIN {X 0,Y 473.965,Z 780.81,A -85,B 0,C 180,E1 13818.105,E2 13818.105} C_VEL
LIN {X 0,Y 473.946,Z 780.81,A -85,B 0,C 180,E1 13824.981,E2 13824.981} C_VEL
LIN {X 0,Y 474.216,Z 780.81,A -85,B 0,C 180,E1 13831.449,E2 13831.449} C_VEL
LIN {X 0,Y 474.378,Z 780.81,A -85,B 0,C 180,E1 13837.528,E2 13837.528} C_VEL
LIN {X 0,Y 474.631,Z 780.81,A -85,B 0,C 180,E1 13843.349,E2 13843.349} C_VEL
LIN {X 0,Y 474.908,Z 780.81,A -85,B 0,C 180,E1 13848.993,E2 13848.993} C_VEL
LIN {X 0,Y 475.19,Z 780.81,A -85,B 0,C 180,E1 13854.524,E2 13854.524} C_VEL
LIN {X 0,Y 475.569,Z 780.81,A -85,B 0,C 180,E1 13859.997,E2 13859.997} C_VEL
LIN {X 0,Y 475.201,Z 780.81,A -85,B 0,C 180,E1 13865.47,E2 13865.47} C_VEL
LIN {X 0,Y 474.922,Z 780.81,A -85,B 0,C 180,E1 13871.001,E2 13871.001} C_VEL
LIN {X 0,Y 474.643,Z 780.81,A -85,B 0,C 180,E1 13877.231,E2 13877.231} C_VEL
LIN {X 0,Y 474.389,Z 780.81,A -85,B 0,C 180,E1 13882.516,E2 13882.516} C_VEL
LIN {X 0,Y 474.245,Z 780.81,A -85,B 0,C 180,E1 13888.543,E2 13888.543} C_VEL
LIN {X 0,Y 474.044,Z 780.81,A -85,B 0,C 180,E1 13895.004,E2 13895.004} C_VEL
LIN {X 0,Y 474.009,Z 780.987,A -85,B 0,C 180,E1 13898.442,E2 13898.442} C_VEL
LIN {X 0,Y 476.355,Z 786.475,A -85,B 0,C 180,E1 13898.902,E2 13898.902} C_VEL
LIN {X 0,Y 498.849,Z 822.749,A -85,B 0,C 180,E1 13902.584,E2 13902.584} C_VEL
LIN {X 0,Y 518.022,Z 860.647,A -85,B 0,C 180,E1 13905.708,E2 13905.708} C_VEL
LIN {X 0,Y 524.448,Z 878.035,A -85,B 0,C 180,E1 13906.978,E2 13906.978} C_VEL
LIN {X 0,Y 518.397,Z 923.865,A -85,B 0,C 180,E1 13908.668,E2 13908.668} C_VEL
LIN {X 0,Y 510.672,Z 969.091,A -85,B 0,C 180,E1 13911.173,E2 13911.173} C_VEL
LIN {X 0,Y 502.436,Z 1009.386,A -85,B 0,C 180,E1 13914.277,E2 13914.277} C_VEL
LIN {X 0,Y 494.57,Z 1044.968,A -85,B 0,C 180,E1 13917.934,E2 13917.934} C_VEL
LIN {X 0,Y 487.762,Z 1075.375,A -85,B 0,C 180,E1 13922.002,E2 13922.002} C_VEL
LIN {X 0,Y 482.165,Z 1102.277,A -85,B 0,C 180,E1 13926.691,E2 13926.691} C_VEL
LIN {X 0,Y 478.272,Z 1125.114,A -85,B 0,C 180,E1 13932.057,E2 13932.057} C_VEL
LIN {X 0,Y 476.372,Z 1140.514,A -85,B 0,C 180,E1 13937.17,E2 13937.17} C_VEL
LIN {X 0,Y 475.75,Z 1149.94,A -85,B 0,C 180,E1 13941.781,E2 13941.781} C_VEL
LIN {X 0,Y 475.556,Z 1155.107,A -85,B 0,C 180,E1 13946.355,E2 13946.355} C_VEL
LIN {X 0,Y 475.593,Z 1156.022,A -85,B 0,C 180,E1 13948.042,E2 13948.042} C_VEL
LIN {X 0,Y 473.192,Z 1156.433,A -85,B 0,C 180,E1 13949.593,E2 13949.593} C_VEL
LIN {X 0,Y 467.629,Z 1155.649,A -85,B 0,C 180,E1 13952.192,E2 13952.192} C_VEL
LIN {X 0,Y 467.79,Z 1151.081,A -85,B 0,C 180,E1 13957.423,E2 13957.423} C_VEL
LIN {X 0,Y 468.504,Z 1141.709,A -85,B 0,C 180,E1 13962.574,E2 13962.574} C_VEL
LIN {X 0,Y 470.575,Z 1125.381,A -85,B 0,C 180,E1 13968.244,E2 13968.244} C_VEL
LIN {X 0,Y 474.556,Z 1104.109,A -85,B 0,C 180,E1 13973.454,E2 13973.454} C_VEL
LIN {X 0,Y 480.321,Z 1078.624,A -85,B 0,C 180,E1 13978.157,E2 13978.157} C_VEL
LIN {X 0,Y 488.04,Z 1047.467,A -85,B 0,C 180,E1 13982.545,E2 13982.545} C_VEL
LIN {X 0,Y 497.02,Z 1010.769,A -85,B 0,C 180,E1 13986.452,E2 13986.452} C_VEL
LIN {X 0,Y 506.214,Z 970.156,A -85,B 0,C 180,E1 13989.647,E2 13989.647} C_VEL
LIN {X 0,Y 514.054,Z 928.902,A -85,B 0,C 180,E1 13992.01,E2 13992.01} C_VEL
LIN {X 0,Y 520.454,Z 886.844,A -85,B 0,C 180,E1 13993.689,E2 13993.689} C_VEL
LIN {X 0,Y 520.85,Z 879.001,A -85,B 0,C 180,E1 13993.995,E2 13993.995} C_VEL
LIN {X 0,Y 504.607,Z 843.143,A -85,B 0,C 180,E1 13997.216,E2 13997.216} C_VEL
LIN {X 0,Y 483.466,Z 808.106,A -85,B 0,C 180,E1 14001.034,E2 14001.034} C_VEL
LIN {X 0,Y 468.816,Z 786.785,A -85,B 0,C 180,E1 14003.954,E2 14003.954} C_VEL
LIN {X 0,Y 466.126,Z 781.658,A -85,B 0,C 180,E1 14004.567,E2 14004.567} C_VEL
LIN {X 0,Y 466.069,Z 780.81,A -85,B 0,C 180,E1 14005.326,E2 14005.326} C_VEL
LIN {X 0,Y 466.262,Z 780.81,A -85,B 0,C 180,E1 14011.048,E2 14011.048} C_VEL
LIN {X 0,Y 466.445,Z 780.81,A -85,B 0,C 180,E1 14017.13,E2 14017.13} C_VEL
LIN {X 0,Y 466.716,Z 780.81,A -85,B 0,C 180,E1 14023.064,E2 14023.064} C_VEL
LIN {X 0,Y 466.953,Z 780.81,A -85,B 0,C 180,E1 14028.809,E2 14028.809} C_VEL
LIN {X 0,Y 467.267,Z 780.81,A -85,B 0,C 180,E1 14034.436,E2 14034.436} C_VEL
LIN {X 0,Y 467.656,Z 780.81,A -85,B 0,C 180,E1 14040.003,E2 14040.003} C_VEL
LIN {X 0,Y 467.345,Z 780.81,A -85,B 0,C 180,E1 14045.568,E2 14045.568} C_VEL
LIN {X 0,Y 466.992,Z 780.81,A -85,B 0,C 180,E1 14051.196,E2 14051.196} C_VEL
LIN {X 0,Y 466.75,Z 780.81,A -85,B 0,C 180,E1 14056.94,E2 14056.94} C_VEL
LIN {X 0,Y 466.424,Z 780.81,A -85,B 0,C 180,E1 14062.877,E2 14062.877} C_VEL
LIN {X 0,Y 466.254,Z 780.81,A -85,B 0,C 180,E1 14069.085,E2 14069.085} C_VEL
LIN {X 0,Y 466.173,Z 781.381,A -85,B 0,C 180,E1 14072.896,E2 14072.896} C_VEL
LIN {X 0,Y 468.619,Z 786.562,A -85,B 0,C 180,E1 14073.468,E2 14073.468} C_VEL
LIN {X 0,Y 483.824,Z 808.953,A -85,B 0,C 180,E1 14076.535,E2 14076.535} C_VEL
LIN {X 0,Y 501.831,Z 840.445,A -85,B 0,C 180,E1 14080.148,E2 14080.148} C_VEL
LIN {X 0,Y 516.012,Z 873.489,A -85,B 0,C 180,E1 14083.432,E2 14083.432} C_VEL
LIN {X 0,Y 518.59,Z 882.343,A -85,B 0,C 180,E1 14084.202,E2 14084.202} C_VEL
LIN {X 0,Y 511.027,Z 926.271,A -85,B 0,C 180,E1 14086.403,E2 14086.403} C_VEL
LIN {X 0,Y 502.137,Z 968.224,A -85,B 0,C 180,E1 14089.402,E2 14089.402} C_VEL
LIN {X 0,Y 492.928,Z 1005.681,A -85,B 0,C 180,E1 14093.042,E2 14093.042} C_VEL
LIN {X 0,Y 484.731,Z 1037.503,A -85,B 0,C 180,E1 14097.167,E2 14097.167} C_VEL
LIN {X 0,Y 477.926,Z 1064.131,A -85,B 0,C 180,E1 14101.689,E2 14101.689} C_VEL
LIN {X 0,Y 473.016,Z 1085.46,A -85,B 0,C 180,E1 14106.465,E2 14106.465} C_VEL
LIN {X 0,Y 469.891,Z 1102.675,A -85,B 0,C 180,E1 14111.762,E2 14111.762} C_VEL
LIN {X 0,Y 468.263,Z 1114.231,A -85,B 0,C 180,E1 14116.946,E2 14116.946} C_VEL
LIN {X 0,Y 467.802,Z 1119.568,A -85,B 0,C 180,E1 14120.706,E2 14120.706} C_VEL
LIN {X 0,Y 467.545,Z 1122.78,A -85,B 0,C 180,E1 14126.295,E2 14126.295} C_VEL
LIN {X 0,Y 467.827,Z 1120.631,A -85,B 0,C 180,E1 14131.852,E2 14131.852} C_VEL
LIN {X 0,Y 468.245,Z 1114.707,A -85,B 0,C 180,E1 14136.487,E2 14136.487} C_VEL
LIN {X 0,Y 469.602,Z 1103.599,A -85,B 0,C 180,E1 14141.603,E2 14141.603} C_VEL
LIN {X 0,Y 472.369,Z 1087.185,A -85,B 0,C 180,E1 14146.734,E2 14146.734} C_VEL
LIN {X 0,Y 477.225,Z 1064.543,A -85,B 0,C 180,E1 14151.844,E2 14151.844} C_VEL
LIN {X 0,Y 483.596,Z 1037.889,A -85,B 0,C 180,E1 14156.361,E2 14156.361} C_VEL
LIN {X 0,Y 491.38,Z 1006.352,A -85,B 0,C 180,E1 14160.435,E2 14160.435} C_VEL
LIN {X 0,Y 499.789,Z 969.926,A -85,B 0,C 180,E1 14163.994,E2 14163.994} C_VEL
LIN {X 0,Y 507.88,Z 929.672,A -85,B 0,C 180,E1 14166.917,E2 14166.917} C_VEL
LIN {X 0,Y 514.84,Z 888.216,A -85,B 0,C 180,E1 14169.078,E2 14169.078} C_VEL
LIN {X 0,Y 515.451,Z 879.031,A -85,B 0,C 180,E1 14169.542,E2 14169.542} C_VEL
LIN {X 0,Y 500.069,Z 840.798,A -85,B 0,C 180,E1 14172.966,E2 14172.966} C_VEL
LIN {X 0,Y 480.717,Z 805.056,A -85,B 0,C 180,E1 14176.523,E2 14176.523} C_VEL
LIN {X 0,Y 466.184,Z 782.381,A -85,B 0,C 180,E1 14179.143,E2 14179.143} C_VEL
